// TIA Portal V20 export
// export: Created 2025-12-01T14:57:38.8034744Z, ExportSetting None, DisplayName Totally Integrated Automation Portal, DisplayVersion V20 Update 3, DisplayName TIA Portal Openness, DisplayVersion V20 Update 3, DisplayName TIA Portal Version Control Interface, DisplayVersion V20 Update 3, DisplayName STEP 7 Professional, DisplayVersion V20 Update 3, DisplayName STEP 7 Safety, DisplayVersion V20 Update 2, DisplayName WinCC Basic/Comfort/Advanced, DisplayVersion V20 Update 3, DisplayName WinCC Professional, DisplayVersion V20 Update 3, DisplayName WinCC Unified, DisplayVersion V20 Update 3
FUNCTION_BLOCK "FB75_MesaRodillos_PaletizadorCajasPlastico"   // FB75, LAD
TITLE = Mesa de Rodillos del DesPaletizador de Paletas
{ S7_Optimized_Access := 'FALSE' }
AUTHOR : PALETIZA
FAMILY : FRUTA
NAME : 20161001
VERSION : 1.0
// stored: AutoNumber false, SetENOAutomatically false
   VAR_INPUT
      Mesa : UInt;   // Mesa de la FB
      Error_Tx : Bool;   // Error en el Tx
      EnTension : Bool;   // Existe Tension en la Mesa
      Termico_Tx : Bool;   // Proteccion del Tx
      pHsMx : Bool;   // pHs de la Mesa
      pHsMx_PR1 : Bool;   // pHs de Protrusion de la Mesa. Nota: No existe >> ON
      Avance_Tx : Bool;   // Avance del Tx
      Retroceso_Tx : Bool;   // Retroceso del Tx
      Termico_MElev : Bool;   // Protecion de la Mesa Elevadora
      MElev_Abajo : Bool;   // Pos. Abajo >>> Mesa Elevadora
      MElev_Paleta : Bool;   // Pos. Paleta Normal >>> Mesa Elevadora
      MElev_EspacioBanda : Bool;   // Pos. Libre para mover la Banda >>> Mesa Elevadora
      ELEV_Bamper : Bool;   // Bamber >>> Mesa Elevadora
      MElev_EnMovimiento : Bool;   // En Movimiento >>> Mesa Elevadora
      PalaFija_IN : Bool;   // Pos. Cerrada >>> Pala Fija (Extendida)
      PalaFija_OUT : Bool;   // Pos. Abierta >>> Pala Fija (Recogida)
      PalaFija_EnMovimiento : Bool;   // En Movimiento >>> Pala Fija
      PalaMovil_IN : Bool;   // Pos. Cerrada >>> Pala Movil (Extendida)
      PalaMovil_OUT : Bool;   // Pos. Abierta >>> Pala Movil (Recogida)
      PalaMovil_EnMovimiento : Bool;   // En Movimiento >>> Pala Movil
      Centrador_IN : Bool;   // Pos. Sacado >>> Centrador
      Centrador_OUT : Bool;   // Pos. Recogido >>> Centrador
      Centrador_EnMovimiento : Bool;   // En Movimiento >>> Centrador
      Aviso_Paletizado : Bool;   // Aviso Paletizar >> Interlock Banda
      PermisoCierrePalas : Bool;   // Permiso Cierre de Palas >> Interlock Banda
      Permitir_AbrirPalas : Bool;   // Permiso DesPaletizar >> Interlock Banda
      Permitir_CerrarPalas : Bool;   // Permiso Abrir Palas >> Interlock Banda
      Permitir_AbrirCentrado : Bool;   // Permiso Abrir Centrador
      Permitir_CerrarCentrado : Bool;   // Permiso Cerrar Centrador
      MAnt_DescargaAct : Bool;   // E1 >> Mesa Anterior DescargaAct
      AVTF_MAnt_Mx : Bool;   // E1 >> Mesa Anterior AVTF
      P_Mens_MAnt_Mx : Bool;   // E1 >> Mesa Anterior P_Mens
      PTF_Mx_MSig : Bool;   // S1 >> Mesa Siguiente PTF
      FTF_Mx_MSig : Bool;   // S1 >> Mesa Siguiente FTF
      MSig_CargaAct : Bool;
      Mx_SimultaneoPaletizado : Bool;   // Config para Simultaneo de Paletizado
      Mx_VelocidadLenta_In : Bool;   // Forzar a Velociada Lenta
      F_EnvMens_Mx : Bool;   // Fin de Envio de Mensaje
      OrdSal_S01 : Bool;   // Orden de Salida por S1 (Paleta Cargada)
      V_CNT_pHsMx : Int := 500;   // Valor de Presencia
      V_CNTSeg_pHsMx : Int := 2000;   // Valor de Seguriadad para Presencia
      V_CNT_PasoLenta : Int := 2000;   // Valor de Paso a Lenta
      V_CNT_ApHsMx : Int := 500;   // Valor de Ausencia
      V_CNTSeg_ApHsMx : Int := 2000;   // Valor de Seguriadad para Ausencia
      V_TMP_EstablePalaMovil_IN : Int := 2000;   // TMP de Estabilidad de Pala Movil Extendida
      V_TOut_Tx_Mx : Int := 15000;   // TimeOut de Entrada por E1
      V_TOut_Palas : Int := 5000;   // TimeOut de las Palas
      V_TOut_Centrado : Int := 5000;   // TimeOut del Centrado
      V_TOut_MElevadora : Int := 10000;   // TimeOut de la Mesa Elevadora
      V_TMP_Protrusion : Int := 200;   // TMP de Protrusion
      V_CNT_PerdidapHs : Int := 1000;   // CNT de Perdida de pHs
   END_VAR
   VAR_OUTPUT
      P_EnvMens_PMx : Bool;   // Permiso de Enviar Mensaje de Presencia
      P_RecepOK_Mx : Bool;   // Recepcion OK
      Permiso_Paletizado : Bool;   // Permiso Paletizar >> Interlock Banda
      FinCierre_Palas : Bool;   // Fin Cierre Palas >> Interlock Banda
      PTF_MAnt_Mx : Bool;   // E1 >> Mesa Anterior PTF
      FTF_MAnt_Mx : Bool;   // E1 >> Mesa Anterior FTF
      AVTF_Mx_MSig : Bool;   // S1 >> Mesa Siguiente AVTF
      P_Mens_Mx_MSig : Bool;   // S1 >> Mesa Siguiente P_Mens
   END_VAR
   VAR
      Anular_prE1 : Bool;   // ???
      Anular_prS3 : Bool;   // ???
      Mx_ET00 : Bool;
      Mx_ET01 : Bool;
      Mx_ET02 : Bool;
      Mx_ET08 : Bool;
      Mx_ET09 : Bool;
      Mx_ET10 : Bool;
      Mx_ET11 : Bool;
      Mx_ET12 : Bool;
      Mx_ET13 : Bool;
      Mx_ET110 : Bool;
      Mx_ET111 : Bool;
      Mx_ET50 : Bool;
      Mx_ET51 : Bool;
      Mx_ET150 : Bool;
      Mx_ET151 : Bool;
      Mx_ET60 : Bool;
      Mx_ET61 : Bool;
      Mx_ET62 : Bool;
      Mx_ET63 : Bool;
      ProtocoloIniciado : Bool;   // Iniciado el Envio del Mensaje de Presencia
      PosMesa_OK : Bool;   // Posicion OK de la Mesa Elevadora
      SimultaneoPaletizado : Bool;   // Simultaneo Realizandose en el Paletizado
      Activar_OperativaPaletizado : Bool;   // Activar la Opertaiva de Simultaneo en el Paletizado
      CNT_pHsMx { S7_SetPoint := 'True'} : "FB910_CNT_UHS";   // CNT de la Presencia
      CNTSeg_pHsMx { S7_SetPoint := 'True'} : "FB910_CNT_UHS";   // CNT de Seguridad de la Presencia
      CNT_ApHsMx { S7_SetPoint := 'True'} : "FB910_CNT_UHS";   // CNT de la Ausencia
      CNTSeg_ApHsMx { S7_SetPoint := 'True'} : "FB910_CNT_UHS";   // CNT de Seguridad de la Ausencia
      TMP_EstablePalaMovil_IN { S7_SetPoint := 'True'} : "FB910_CNT_UHS";   // TMP de Estabilidad de Pala Movil Extendida
      TMP_EnTension { ExternalAccessible := 'False'; ExternalVisible := 'False'; ExternalWritable := 'False'; S7_SetPoint := 'True'} : "FB910_CNT_UHS";
      TOut_Av_Mx { S7_SetPoint := 'True'} : "FB910_CNT_UHS";   // Time Out de Entrada de E1
      TOut_MElevadora { S7_SetPoint := 'True'} : "FB910_CNT_UHS";   // Time Out de Recigida y Extension del Centrador
      TOut_Centrado { S7_SetPoint := 'True'} : "FB910_CNT_UHS";   // Time Out de Recigida y Extension de Pala Fija
      TOut_PalasFija { S7_SetPoint := 'True'} : "FB910_CNT_UHS";   // Time Out de Recigida y Extension de Pala Movil
      TOut_PalasMovil { S7_SetPoint := 'True'} : "FB910_CNT_UHS";   // Time Out de Subir y Bajar de la Mesa Elevadora
      TMP_Protrusion { S7_SetPoint := 'True'} : "FB910_CNT_UHS";   // TMP de la Protrusion
      CNT_PerdidapHs { S7_SetPoint := 'True'} : "FB910_CNT_UHS";   // CNT de Perdida de pHs
      STAT_EnvMens_PMx : Bool;   // Interna >> Envio del Mensaje de Presencia
      STAT_FTF_MAnt_Mx : Bool;   // Interna >> FTF de MAnt >> Mx
      STAT_AVTF_Mx_MSig : Bool;   // Interna >> AVTF de Mx >> MSig
      MA_Cerrar_Centrado : Bool;   // ????
      MA_Abrir_Centrado : Bool;   // ????
      MA_Abrir_PalasMovil : Bool;   // ????
      MA_Cerrar_PalasMovil : Bool;   // ????
      MA_Abrir_PalasFija : Bool;   // ????
      MA_Cerrar_PalasFija : Bool;   // ????
   END_VAR
   VAR_TEMP
      EstadoZona : "EstadoZona";   // Estado de Zona de la Mesa
      EstadoVI : "EstadosMesa";   // Estado del Vehiculo Inteliguente de la Mesa
      EstadoMAQ : "EstadoMaquina_MesaRodillos_PaletizadorCajasPlastico";   // Estado del Vehiculo Inteliguente de la Maquina
      ConfigFB : "UDT_ConfigFB";   // Configuracion de la FB de la Mesa
      V_Protrusion : Int;
      Aux_ET00 : Bool;
   END_VAR
BEGIN

REGION Network 1: Configuraciones Especiales
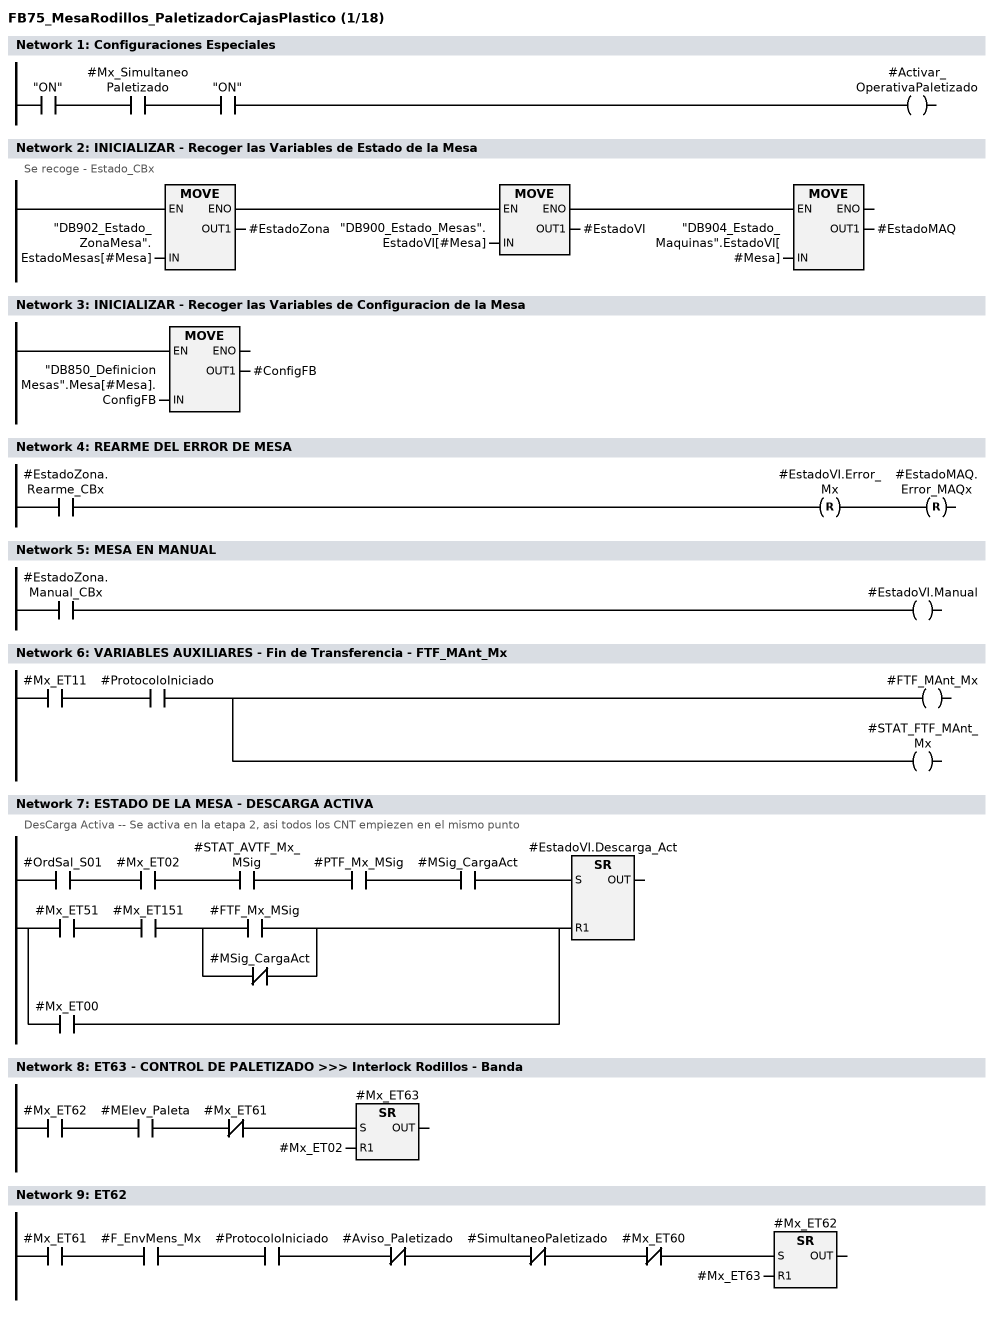
   RUNG wire#powerrail
      Contact( "ON" )
      Contact( #Mx_SimultaneoPaletizado )
      Contact( "ON" )
      Coil( #Activar_OperativaPaletizado )
   END_RUNG
   // the same network as SCL:
   #Activar_OperativaPaletizado := "ON" AND #Mx_SimultaneoPaletizado AND "ON";
END_REGION

REGION Network 2: INICIALIZAR - Recoger las Variables de Estado de la Mesa
   // Se recoge - Estado_CBx
   RUNG wire#powerrail
      Move(in := "DB902_Estado_ZonaMesa".EstadoMesas[#Mesa], out1 => #EstadoZona)
      Move(in := "DB900_Estado_Mesas".EstadoVI[#Mesa], out1 => #EstadoVI)
      Move(in := "DB904_Estado_Maquinas".EstadoVI[#Mesa], out1 => #EstadoMAQ)
   END_RUNG
   // the same network as SCL:
   #EstadoZona := "DB902_Estado_ZonaMesa".EstadoMesas[#Mesa];
   #EstadoVI := "DB900_Estado_Mesas".EstadoVI[#Mesa];
   #EstadoMAQ := "DB904_Estado_Maquinas".EstadoVI[#Mesa];
END_REGION

REGION Network 3: INICIALIZAR - Recoger las Variables de Configuracion de la Mesa
   RUNG wire#powerrail
      Move(in := "DB850_DefinicionMesas".Mesa[#Mesa].ConfigFB, out1 => #ConfigFB)
   END_RUNG
   // the same network as SCL:
   #ConfigFB := "DB850_DefinicionMesas".Mesa[#Mesa].ConfigFB;
END_REGION

REGION Network 4: REARME DEL ERROR DE MESA
   RUNG wire#powerrail
      Contact( #EstadoZona.Rearme_CBx )
      R_Coil( #EstadoVI.Error_Mx )
      R_Coil( #EstadoMAQ.Error_MAQx )
   END_RUNG
   // the same network as SCL:
   IF #EstadoZona.Rearme_CBx THEN
       #EstadoVI.Error_Mx := FALSE;
       #EstadoMAQ.Error_MAQx := FALSE;
   END_IF;
END_REGION

REGION Network 5: MESA EN MANUAL
   RUNG wire#powerrail
      Contact( #EstadoZona.Manual_CBx )
      Coil( #EstadoVI.Manual )
   END_RUNG
   // the same network as SCL:
   #EstadoVI.Manual := #EstadoZona.Manual_CBx;
END_REGION

REGION Network 6: VARIABLES AUXILIARES - Fin de Transferencia - FTF_MAnt_Mx
   RUNG wire#powerrail
      Contact( #Mx_ET11 )
      Contact( #ProtocoloIniciado )
      wire#w1
      Coil( #FTF_MAnt_Mx )
   END_RUNG
   RUNG wire#w1
      Coil( #STAT_FTF_MAnt_Mx )
   END_RUNG
   // the same network as SCL:
   #FTF_MAnt_Mx := #Mx_ET11 AND #ProtocoloIniciado;
   #STAT_FTF_MAnt_Mx := #FTF_MAnt_Mx;
END_REGION

REGION Network 7: ESTADO DE LA MESA - DESCARGA ACTIVA
   // DesCarga Activa -- Se activa en la etapa 2, asi todos los CNT empiezen en el mismo punto
   RUNG wire#powerrail
      Contact( #OrdSal_S01 )
      Contact( #Mx_ET02 )
      Contact( #STAT_AVTF_Mx_MSig )
      Contact( #PTF_Mx_MSig )
      Contact( #MSig_CargaAct )
      S_SR(operand := #EstadoVI.Descarga_Act, r1 := wire#w2)
   END_RUNG
   RUNG wire#powerrail
      Contact( #Mx_ET51 )
      Contact( #Mx_ET151 )
      wire#w1
      Contact( #FTF_Mx_MSig )
   END_RUNG wire#w2
   RUNG wire#w1
      I_Contact( #MSig_CargaAct )
   END_RUNG wire#w2
   RUNG wire#powerrail
      Contact( #Mx_ET00 )
   END_RUNG wire#w2
   // the same network as SCL:
   IF #OrdSal_S01 AND #Mx_ET02 AND #STAT_AVTF_Mx_MSig AND #PTF_Mx_MSig AND #MSig_CargaAct THEN
       #EstadoVI.Descarga_Act := TRUE;   // SR flip-flop
   END_IF;
   IF (#Mx_ET51 AND #Mx_ET151 AND (#FTF_Mx_MSig OR NOT #MSig_CargaAct)) OR #Mx_ET00 THEN
       #EstadoVI.Descarga_Act := FALSE;
   END_IF;
END_REGION

REGION Network 8: ET63 - CONTROL DE PALETIZADO >>> Interlock Rodillos - Banda
   RUNG wire#powerrail
      Contact( #Mx_ET62 )
      Contact( #MElev_Paleta )
      I_Contact( #Mx_ET61 )
      S_SR(operand := #Mx_ET63, r1 := #Mx_ET02)
   END_RUNG
   // the same network as SCL:
   IF #Mx_ET62 AND #MElev_Paleta AND NOT #Mx_ET61 THEN
       #Mx_ET63 := TRUE;   // SR flip-flop
   END_IF;
   IF #Mx_ET02 THEN #Mx_ET63 := FALSE; END_IF;
END_REGION

REGION Network 9: ET62
   RUNG wire#powerrail
      Contact( #Mx_ET61 )
      Contact( #F_EnvMens_Mx )
      Contact( #ProtocoloIniciado )
      I_Contact( #Aviso_Paletizado )
      I_Contact( #SimultaneoPaletizado )
      I_Contact( #Mx_ET60 )
      S_SR(operand := #Mx_ET62, r1 := #Mx_ET63)
   END_RUNG
   // the same network as SCL:
   IF #Mx_ET61 AND #F_EnvMens_Mx AND #ProtocoloIniciado AND NOT #Aviso_Paletizado AND NOT #SimultaneoPaletizado AND NOT #Mx_ET60 THEN
       #Mx_ET62 := TRUE;   // SR flip-flop
   END_IF;
   IF #Mx_ET63 THEN #Mx_ET62 := FALSE; END_IF;
END_REGION

REGION Network 10: ET61
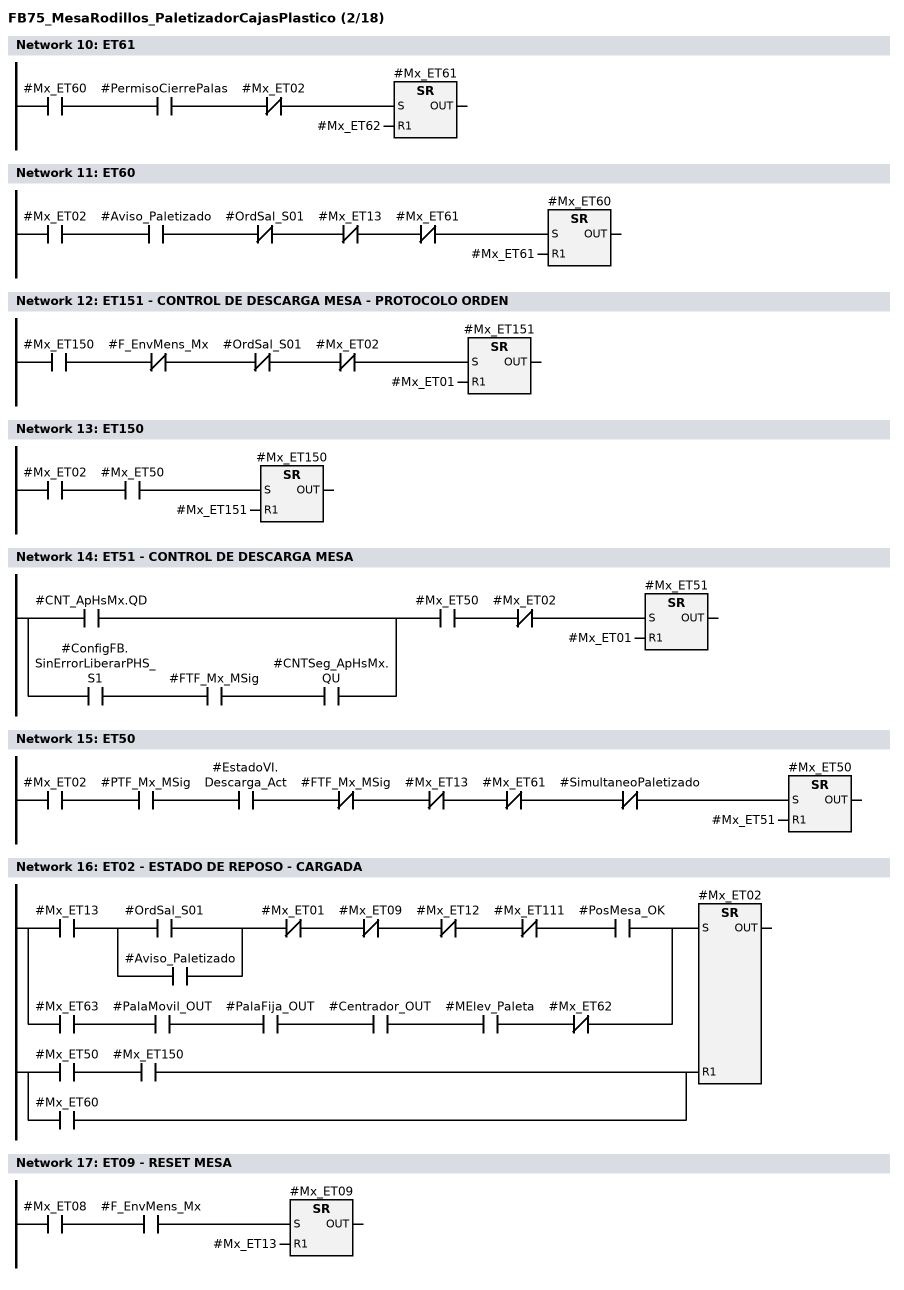
   RUNG wire#powerrail
      Contact( #Mx_ET60 )
      Contact( #PermisoCierrePalas )
      I_Contact( #Mx_ET02 )
      S_SR(operand := #Mx_ET61, r1 := #Mx_ET62)
   END_RUNG
   // the same network as SCL:
   IF #Mx_ET60 AND #PermisoCierrePalas AND NOT #Mx_ET02 THEN
       #Mx_ET61 := TRUE;   // SR flip-flop
   END_IF;
   IF #Mx_ET62 THEN #Mx_ET61 := FALSE; END_IF;
END_REGION

REGION Network 11: ET60
   RUNG wire#powerrail
      Contact( #Mx_ET02 )
      Contact( #Aviso_Paletizado )
      I_Contact( #OrdSal_S01 )
      I_Contact( #Mx_ET13 )
      I_Contact( #Mx_ET61 )
      S_SR(operand := #Mx_ET60, r1 := #Mx_ET61)
   END_RUNG
   // the same network as SCL:
   IF #Mx_ET02 AND #Aviso_Paletizado AND NOT #OrdSal_S01 AND NOT #Mx_ET13 AND NOT #Mx_ET61 THEN
       #Mx_ET60 := TRUE;   // SR flip-flop
   END_IF;
   IF #Mx_ET61 THEN #Mx_ET60 := FALSE; END_IF;
END_REGION

REGION Network 12: ET151 - CONTROL DE DESCARGA MESA - PROTOCOLO ORDEN
   RUNG wire#powerrail
      Contact( #Mx_ET150 )
      I_Contact( #F_EnvMens_Mx )
      I_Contact( #OrdSal_S01 )
      I_Contact( #Mx_ET02 )
      S_SR(operand := #Mx_ET151, r1 := #Mx_ET01)
   END_RUNG
   // the same network as SCL:
   IF #Mx_ET150 AND NOT #F_EnvMens_Mx AND NOT #OrdSal_S01 AND NOT #Mx_ET02 THEN
       #Mx_ET151 := TRUE;   // SR flip-flop
   END_IF;
   IF #Mx_ET01 THEN #Mx_ET151 := FALSE; END_IF;
END_REGION

REGION Network 13: ET150
   RUNG wire#powerrail
      Contact( #Mx_ET02 )
      Contact( #Mx_ET50 )
      S_SR(operand := #Mx_ET150, r1 := #Mx_ET151)
   END_RUNG
   // the same network as SCL:
   IF #Mx_ET02 AND #Mx_ET50 THEN
       #Mx_ET150 := TRUE;   // SR flip-flop
   END_IF;
   IF #Mx_ET151 THEN #Mx_ET150 := FALSE; END_IF;
END_REGION

REGION Network 14: ET51 - CONTROL DE DESCARGA MESA
   RUNG wire#powerrail
      Contact( #CNT_ApHsMx.QD )
      wire#w1
      Contact( #Mx_ET50 )
      I_Contact( #Mx_ET02 )
      S_SR(operand := #Mx_ET51, r1 := #Mx_ET01)
   END_RUNG
   RUNG wire#powerrail
      Contact( #ConfigFB.SinErrorLiberarPHS_S1 )
      Contact( #FTF_Mx_MSig )
      Contact( #CNTSeg_ApHsMx.QU )
   END_RUNG wire#w1
   // the same network as SCL:
   IF (#CNT_ApHsMx.QD OR (#ConfigFB.SinErrorLiberarPHS_S1 AND #FTF_Mx_MSig AND #CNTSeg_ApHsMx.QU)) AND #Mx_ET50 AND NOT #Mx_ET02 THEN
       #Mx_ET51 := TRUE;   // SR flip-flop
   END_IF;
   IF #Mx_ET01 THEN #Mx_ET51 := FALSE; END_IF;
END_REGION

REGION Network 15: ET50
   RUNG wire#powerrail
      Contact( #Mx_ET02 )
      Contact( #PTF_Mx_MSig )
      Contact( #EstadoVI.Descarga_Act )
      I_Contact( #FTF_Mx_MSig )
      I_Contact( #Mx_ET13 )
      I_Contact( #Mx_ET61 )
      I_Contact( #SimultaneoPaletizado )
      S_SR(operand := #Mx_ET50, r1 := #Mx_ET51)
   END_RUNG
   // the same network as SCL:
   IF #Mx_ET02 AND #PTF_Mx_MSig AND #EstadoVI.Descarga_Act AND NOT #FTF_Mx_MSig AND NOT #Mx_ET13 AND NOT #Mx_ET61 AND NOT #SimultaneoPaletizado THEN
       #Mx_ET50 := TRUE;   // SR flip-flop
   END_IF;
   IF #Mx_ET51 THEN #Mx_ET50 := FALSE; END_IF;
END_REGION

REGION Network 16: ET02 - ESTADO DE REPOSO - CARGADA
   RUNG wire#powerrail
      Contact( #Mx_ET13 )
      wire#w1
      Contact( #OrdSal_S01 )
      wire#w2
      I_Contact( #Mx_ET01 )
      I_Contact( #Mx_ET09 )
      I_Contact( #Mx_ET12 )
      I_Contact( #Mx_ET111 )
      Contact( #PosMesa_OK )
      wire#w3
      S_SR(operand := #Mx_ET02, r1 := wire#w4)
   END_RUNG
   RUNG wire#w1
      Contact( #Aviso_Paletizado )
   END_RUNG wire#w2
   RUNG wire#powerrail
      Contact( #Mx_ET63 )
      Contact( #PalaMovil_OUT )
      Contact( #PalaFija_OUT )
      Contact( #Centrador_OUT )
      Contact( #MElev_Paleta )
      I_Contact( #Mx_ET62 )
   END_RUNG wire#w3
   RUNG wire#powerrail
      Contact( #Mx_ET50 )
      Contact( #Mx_ET150 )
   END_RUNG wire#w4
   RUNG wire#powerrail
      Contact( #Mx_ET60 )
   END_RUNG wire#w4
   // the same network as SCL:
   IF (#Mx_ET13 AND (#OrdSal_S01 OR #Aviso_Paletizado) AND NOT #Mx_ET01 AND NOT #Mx_ET09 AND NOT #Mx_ET12 AND NOT #Mx_ET111 AND #PosMesa_OK) OR (#Mx_ET63 AND #PalaMovil_OUT AND #PalaFija_OUT AND #Centrador_OUT AND #MElev_Paleta AND NOT #Mx_ET62) THEN
       #Mx_ET02 := TRUE;   // SR flip-flop
   END_IF;
   IF (#Mx_ET50 AND #Mx_ET150) OR #Mx_ET60 THEN #Mx_ET02 := FALSE; END_IF;
END_REGION

REGION Network 17: ET09 - RESET MESA
   RUNG wire#powerrail
      Contact( #Mx_ET08 )
      Contact( #F_EnvMens_Mx )
      S_SR(operand := #Mx_ET09, r1 := #Mx_ET13)
   END_RUNG
   // the same network as SCL:
   IF #Mx_ET08 AND #F_EnvMens_Mx THEN
       #Mx_ET09 := TRUE;   // SR flip-flop
   END_IF;
   IF #Mx_ET13 THEN #Mx_ET09 := FALSE; END_IF;
END_REGION

REGION Network 18: ET08
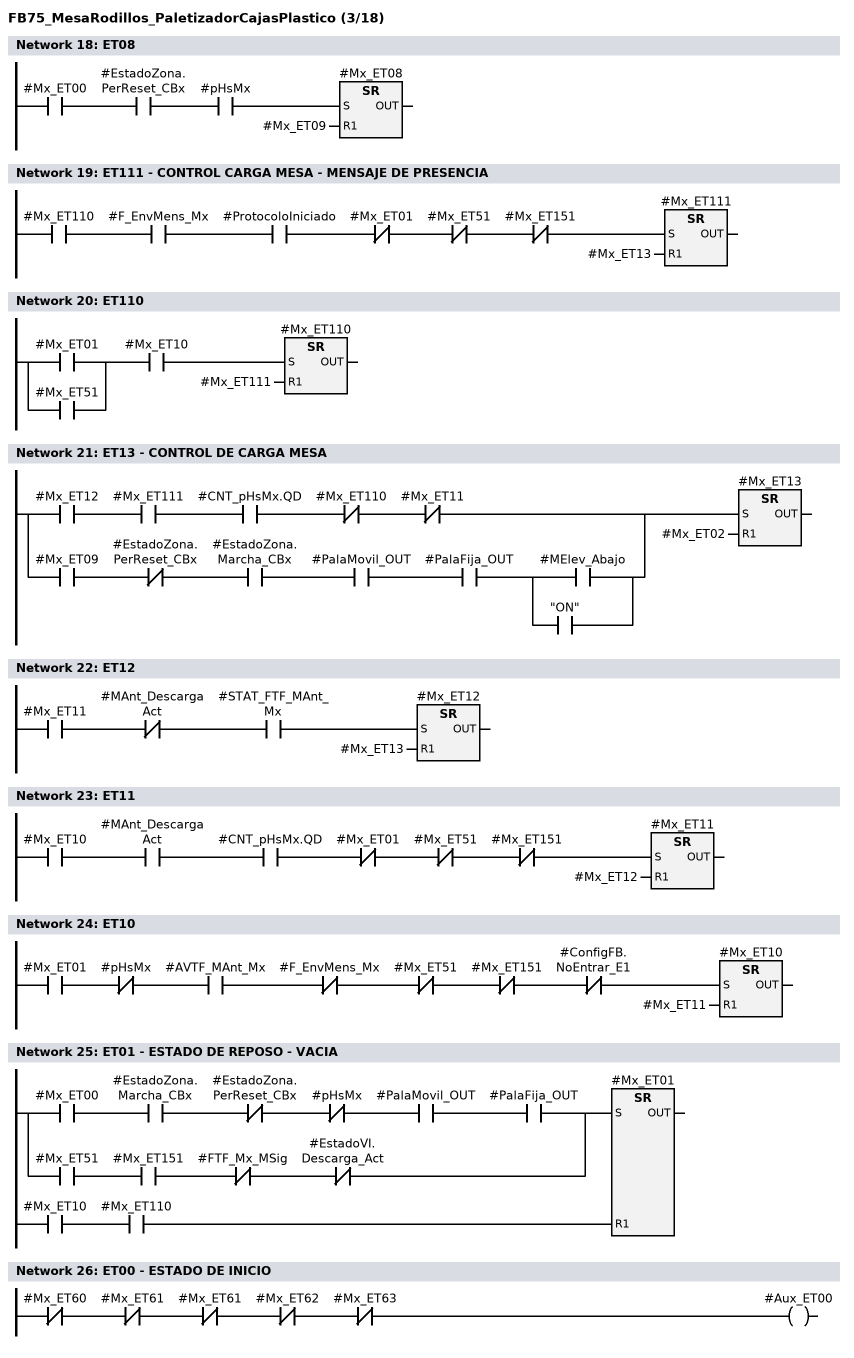
   RUNG wire#powerrail
      Contact( #Mx_ET00 )
      Contact( #EstadoZona.PerReset_CBx )
      Contact( #pHsMx )
      S_SR(operand := #Mx_ET08, r1 := #Mx_ET09)
   END_RUNG
   // the same network as SCL:
   IF #Mx_ET00 AND #EstadoZona.PerReset_CBx AND #pHsMx THEN
       #Mx_ET08 := TRUE;   // SR flip-flop
   END_IF;
   IF #Mx_ET09 THEN #Mx_ET08 := FALSE; END_IF;
END_REGION

REGION Network 19: ET111 - CONTROL CARGA MESA - MENSAJE DE PRESENCIA
   RUNG wire#powerrail
      Contact( #Mx_ET110 )
      Contact( #F_EnvMens_Mx )
      Contact( #ProtocoloIniciado )
      I_Contact( #Mx_ET01 )
      I_Contact( #Mx_ET51 )
      I_Contact( #Mx_ET151 )
      S_SR(operand := #Mx_ET111, r1 := #Mx_ET13)
   END_RUNG
   // the same network as SCL:
   IF #Mx_ET110 AND #F_EnvMens_Mx AND #ProtocoloIniciado AND NOT #Mx_ET01 AND NOT #Mx_ET51 AND NOT #Mx_ET151 THEN
       #Mx_ET111 := TRUE;   // SR flip-flop
   END_IF;
   IF #Mx_ET13 THEN #Mx_ET111 := FALSE; END_IF;
END_REGION

REGION Network 20: ET110
   RUNG wire#powerrail
      Contact( #Mx_ET01 )
      wire#w1
      Contact( #Mx_ET10 )
      S_SR(operand := #Mx_ET110, r1 := #Mx_ET111)
   END_RUNG
   RUNG wire#powerrail
      Contact( #Mx_ET51 )
   END_RUNG wire#w1
   // the same network as SCL:
   IF (#Mx_ET01 OR #Mx_ET51) AND #Mx_ET10 THEN
       #Mx_ET110 := TRUE;   // SR flip-flop
   END_IF;
   IF #Mx_ET111 THEN #Mx_ET110 := FALSE; END_IF;
END_REGION

REGION Network 21: ET13 - CONTROL DE CARGA MESA
   RUNG wire#powerrail
      Contact( #Mx_ET12 )
      Contact( #Mx_ET111 )
      Contact( #CNT_pHsMx.QD )
      I_Contact( #Mx_ET110 )
      I_Contact( #Mx_ET11 )
      wire#w1
      S_SR(operand := #Mx_ET13, r1 := #Mx_ET02)
   END_RUNG
   RUNG wire#powerrail
      Contact( #Mx_ET09 )
      I_Contact( #EstadoZona.PerReset_CBx )
      Contact( #EstadoZona.Marcha_CBx )
      Contact( #PalaMovil_OUT )
      Contact( #PalaFija_OUT )
      wire#w2
      Contact( #MElev_Abajo )
   END_RUNG wire#w1
   RUNG wire#w2
      Contact( "ON" )
   END_RUNG wire#w1
   // the same network as SCL:
   IF (#Mx_ET12 AND #Mx_ET111 AND #CNT_pHsMx.QD AND NOT #Mx_ET110 AND NOT #Mx_ET11) OR (#Mx_ET09 AND NOT #EstadoZona.PerReset_CBx AND #EstadoZona.Marcha_CBx AND #PalaMovil_OUT AND #PalaFija_OUT AND (#MElev_Abajo OR "ON")) THEN
       #Mx_ET13 := TRUE;   // SR flip-flop
   END_IF;
   IF #Mx_ET02 THEN #Mx_ET13 := FALSE; END_IF;
END_REGION

REGION Network 22: ET12
   RUNG wire#powerrail
      Contact( #Mx_ET11 )
      I_Contact( #MAnt_DescargaAct )
      Contact( #STAT_FTF_MAnt_Mx )
      S_SR(operand := #Mx_ET12, r1 := #Mx_ET13)
   END_RUNG
   // the same network as SCL:
   IF #Mx_ET11 AND NOT #MAnt_DescargaAct AND #STAT_FTF_MAnt_Mx THEN
       #Mx_ET12 := TRUE;   // SR flip-flop
   END_IF;
   IF #Mx_ET13 THEN #Mx_ET12 := FALSE; END_IF;
END_REGION

REGION Network 23: ET11
   RUNG wire#powerrail
      Contact( #Mx_ET10 )
      Contact( #MAnt_DescargaAct )
      Contact( #CNT_pHsMx.QD )
      I_Contact( #Mx_ET01 )
      I_Contact( #Mx_ET51 )
      I_Contact( #Mx_ET151 )
      S_SR(operand := #Mx_ET11, r1 := #Mx_ET12)
   END_RUNG
   // the same network as SCL:
   IF #Mx_ET10 AND #MAnt_DescargaAct AND #CNT_pHsMx.QD AND NOT #Mx_ET01 AND NOT #Mx_ET51 AND NOT #Mx_ET151 THEN
       #Mx_ET11 := TRUE;   // SR flip-flop
   END_IF;
   IF #Mx_ET12 THEN #Mx_ET11 := FALSE; END_IF;
END_REGION

REGION Network 24: ET10
   RUNG wire#powerrail
      Contact( #Mx_ET01 )
      I_Contact( #pHsMx )
      Contact( #AVTF_MAnt_Mx )
      I_Contact( #F_EnvMens_Mx )
      I_Contact( #Mx_ET51 )
      I_Contact( #Mx_ET151 )
      I_Contact( #ConfigFB.NoEntrar_E1 )
      S_SR(operand := #Mx_ET10, r1 := #Mx_ET11)
   END_RUNG
   // the same network as SCL:
   IF #Mx_ET01 AND NOT #pHsMx AND #AVTF_MAnt_Mx AND NOT #F_EnvMens_Mx AND NOT #Mx_ET51 AND NOT #Mx_ET151 AND NOT #ConfigFB.NoEntrar_E1 THEN
       #Mx_ET10 := TRUE;   // SR flip-flop
   END_IF;
   IF #Mx_ET11 THEN #Mx_ET10 := FALSE; END_IF;
END_REGION

REGION Network 25: ET01 - ESTADO DE REPOSO - VACIA
   RUNG wire#powerrail
      Contact( #Mx_ET00 )
      Contact( #EstadoZona.Marcha_CBx )
      I_Contact( #EstadoZona.PerReset_CBx )
      I_Contact( #pHsMx )
      Contact( #PalaMovil_OUT )
      Contact( #PalaFija_OUT )
      wire#w1
      S_SR(operand := #Mx_ET01, r1 := wire#w2)
   END_RUNG
   RUNG wire#powerrail
      Contact( #Mx_ET51 )
      Contact( #Mx_ET151 )
      I_Contact( #FTF_Mx_MSig )
      I_Contact( #EstadoVI.Descarga_Act )
   END_RUNG wire#w1
   RUNG wire#powerrail
      Contact( #Mx_ET10 )
      Contact( #Mx_ET110 )
   END_RUNG wire#w2
   // the same network as SCL:
   IF (#Mx_ET00 AND #EstadoZona.Marcha_CBx AND NOT #EstadoZona.PerReset_CBx AND NOT #pHsMx AND #PalaMovil_OUT AND #PalaFija_OUT) OR (#Mx_ET51 AND #Mx_ET151 AND NOT #FTF_Mx_MSig AND NOT #EstadoVI.Descarga_Act) THEN
       #Mx_ET01 := TRUE;   // SR flip-flop
   END_IF;
   IF #Mx_ET10 AND #Mx_ET110 THEN #Mx_ET01 := FALSE; END_IF;
END_REGION

REGION Network 26: ET00 - ESTADO DE INICIO
   RUNG wire#powerrail
      I_Contact( #Mx_ET60 )
      I_Contact( #Mx_ET61 )
      I_Contact( #Mx_ET61 )
      I_Contact( #Mx_ET62 )
      I_Contact( #Mx_ET63 )
      Coil( #Aux_ET00 )
   END_RUNG
   // the same network as SCL:
   #Aux_ET00 := NOT #Mx_ET60 AND NOT #Mx_ET61 AND NOT #Mx_ET61 AND NOT #Mx_ET62 AND NOT #Mx_ET63;
END_REGION

REGION Network 27: ---
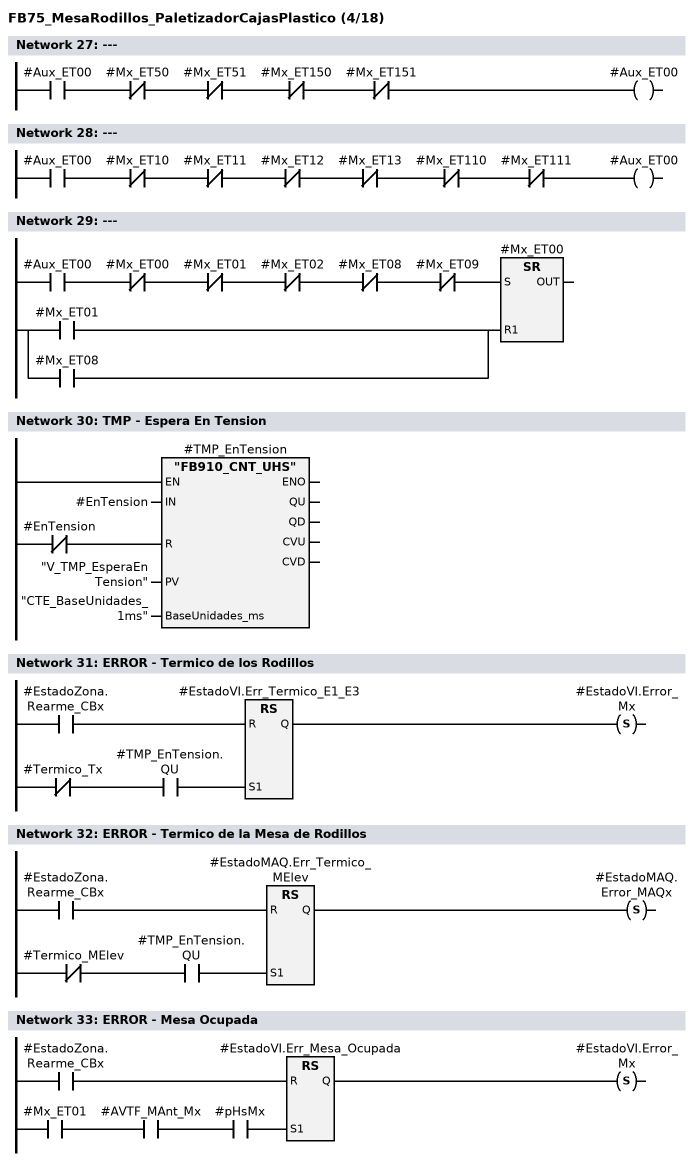
   RUNG wire#powerrail
      Contact( #Aux_ET00 )
      I_Contact( #Mx_ET50 )
      I_Contact( #Mx_ET51 )
      I_Contact( #Mx_ET150 )
      I_Contact( #Mx_ET151 )
      Coil( #Aux_ET00 )
   END_RUNG
   // the same network as SCL:
   #Aux_ET00 := #Aux_ET00 AND NOT #Mx_ET50 AND NOT #Mx_ET51 AND NOT #Mx_ET150 AND NOT #Mx_ET151;
END_REGION

REGION Network 28: ---
   RUNG wire#powerrail
      Contact( #Aux_ET00 )
      I_Contact( #Mx_ET10 )
      I_Contact( #Mx_ET11 )
      I_Contact( #Mx_ET12 )
      I_Contact( #Mx_ET13 )
      I_Contact( #Mx_ET110 )
      I_Contact( #Mx_ET111 )
      Coil( #Aux_ET00 )
   END_RUNG
   // the same network as SCL:
   #Aux_ET00 := #Aux_ET00 AND NOT #Mx_ET10 AND NOT #Mx_ET11 AND NOT #Mx_ET12 AND NOT #Mx_ET13 AND NOT #Mx_ET110 AND NOT #Mx_ET111;
END_REGION

REGION Network 29: ---
   RUNG wire#powerrail
      Contact( #Aux_ET00 )
      I_Contact( #Mx_ET00 )
      I_Contact( #Mx_ET01 )
      I_Contact( #Mx_ET02 )
      I_Contact( #Mx_ET08 )
      I_Contact( #Mx_ET09 )
      S_SR(operand := #Mx_ET00, r1 := wire#w1)
   END_RUNG
   RUNG wire#powerrail
      Contact( #Mx_ET01 )
   END_RUNG wire#w1
   RUNG wire#powerrail
      Contact( #Mx_ET08 )
   END_RUNG wire#w1
   // the same network as SCL:
   IF #Aux_ET00 AND NOT #Mx_ET00 AND NOT #Mx_ET01 AND NOT #Mx_ET02 AND NOT #Mx_ET08 AND NOT #Mx_ET09 THEN
       #Mx_ET00 := TRUE;   // SR flip-flop
   END_IF;
   IF #Mx_ET01 OR #Mx_ET08 THEN #Mx_ET00 := FALSE; END_IF;
END_REGION

REGION Network 30: TMP - Espera En Tension
   RUNG wire#powerrail
      #TMP_EnTension(R := wire#w1, IN := #EnTension, PV := "V_TMP_EsperaEnTension", BaseUnidades_ms := "CTE_BaseUnidades_1ms", QU =>, QD =>, CVU =>, CVD =>)
   END_RUNG
   RUNG wire#powerrail
      I_Contact( #EnTension )
   END_RUNG wire#w1
   // the same network as SCL:
   #TMP_EnTension(IN := #EnTension,   // "FB910_CNT_UHS"
                  R := NOT #EnTension,
                  PV := "V_TMP_EsperaEnTension",
                  BaseUnidades_ms := "CTE_BaseUnidades_1ms");
END_REGION

REGION Network 31: ERROR - Termico de los Rodillos
   RUNG wire#powerrail
      Contact( #EstadoZona.Rearme_CBx )
      S_RS(operand := #EstadoVI.Err_Termico_E1_E3, s1 := wire#w1)
      S_Coil( #EstadoVI.Error_Mx )
   END_RUNG
   RUNG wire#powerrail
      I_Contact( #Termico_Tx )
      Contact( #TMP_EnTension.QU )
   END_RUNG wire#w1
   // the same network as SCL:
   IF #EstadoZona.Rearme_CBx THEN
       #EstadoVI.Err_Termico_E1_E3 := FALSE;   // RS flip-flop
   END_IF;
   IF NOT #Termico_Tx AND #TMP_EnTension.QU THEN #EstadoVI.Err_Termico_E1_E3 := TRUE; END_IF;
   IF #EstadoVI.Err_Termico_E1_E3 THEN #EstadoVI.Error_Mx := TRUE; END_IF;
END_REGION

REGION Network 32: ERROR - Termico de la Mesa de Rodillos
   RUNG wire#powerrail
      Contact( #EstadoZona.Rearme_CBx )
      S_RS(operand := #EstadoMAQ.Err_Termico_MElev, s1 := wire#w1)
      S_Coil( #EstadoMAQ.Error_MAQx )
   END_RUNG
   RUNG wire#powerrail
      I_Contact( #Termico_MElev )
      Contact( #TMP_EnTension.QU )
   END_RUNG wire#w1
   // the same network as SCL:
   IF #EstadoZona.Rearme_CBx THEN
       #EstadoMAQ.Err_Termico_MElev := FALSE;   // RS flip-flop
   END_IF;
   IF NOT #Termico_MElev AND #TMP_EnTension.QU THEN #EstadoMAQ.Err_Termico_MElev := TRUE; END_IF;
   IF #EstadoMAQ.Err_Termico_MElev THEN #EstadoMAQ.Error_MAQx := TRUE; END_IF;
END_REGION

REGION Network 33: ERROR - Mesa Ocupada
   RUNG wire#powerrail
      Contact( #EstadoZona.Rearme_CBx )
      S_RS(operand := #EstadoVI.Err_Mesa_Ocupada, s1 := wire#w1)
      S_Coil( #EstadoVI.Error_Mx )
   END_RUNG
   RUNG wire#powerrail
      Contact( #Mx_ET01 )
      Contact( #AVTF_MAnt_Mx )
      Contact( #pHsMx )
   END_RUNG wire#w1
   // the same network as SCL:
   IF #EstadoZona.Rearme_CBx THEN
       #EstadoVI.Err_Mesa_Ocupada := FALSE;   // RS flip-flop
   END_IF;
   IF #Mx_ET01 AND #AVTF_MAnt_Mx AND #pHsMx THEN #EstadoVI.Err_Mesa_Ocupada := TRUE; END_IF;
   IF #EstadoVI.Err_Mesa_Ocupada THEN #EstadoVI.Error_Mx := TRUE; END_IF;
END_REGION

REGION Network 34: CNT - ERROR - Arrastre
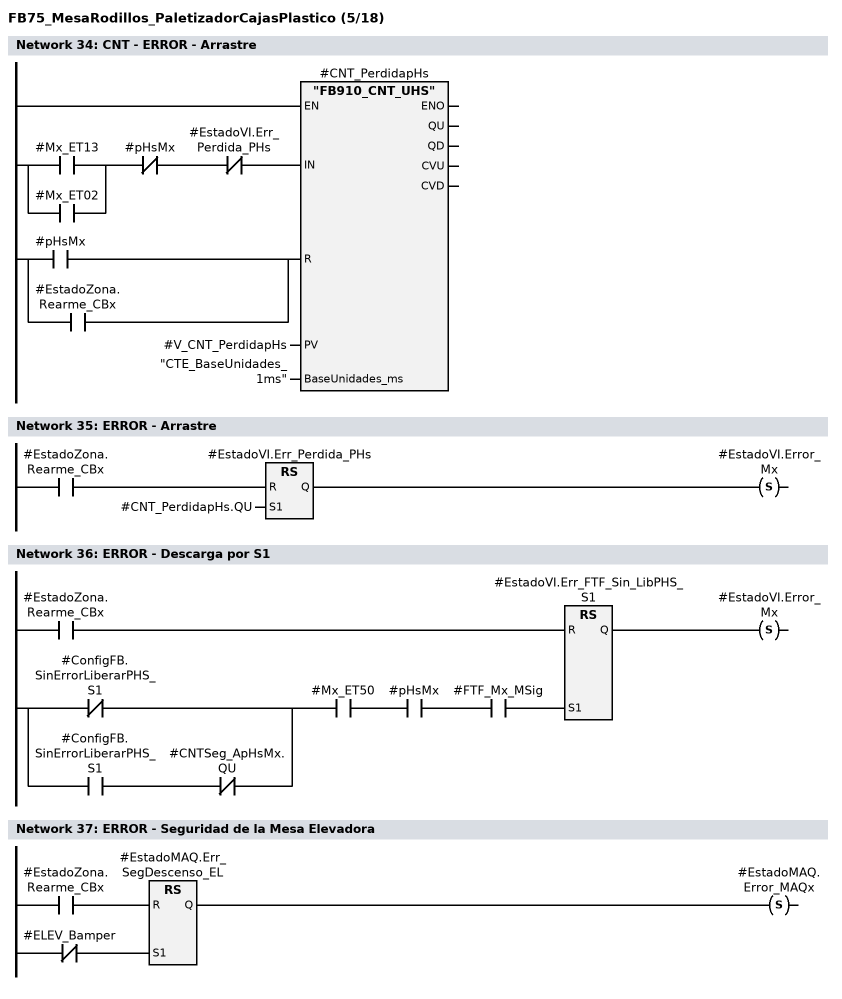
   RUNG wire#powerrail
      #CNT_PerdidapHs(IN := wire#w2, R := wire#w3, PV := #V_CNT_PerdidapHs, BaseUnidades_ms := "CTE_BaseUnidades_1ms", QU =>, QD =>, CVU =>, CVD =>)
   END_RUNG
   RUNG wire#powerrail
      Contact( #Mx_ET13 )
      wire#w1
      I_Contact( #pHsMx )
      I_Contact( #EstadoVI.Err_Perdida_PHs )
   END_RUNG wire#w2
   RUNG wire#powerrail
      Contact( #Mx_ET02 )
   END_RUNG wire#w1
   RUNG wire#powerrail
      Contact( #pHsMx )
   END_RUNG wire#w3
   RUNG wire#powerrail
      Contact( #EstadoZona.Rearme_CBx )
   END_RUNG wire#w3
   // the same network as SCL:
   #CNT_PerdidapHs(IN := (#Mx_ET13 OR #Mx_ET02) AND NOT #pHsMx AND NOT #EstadoVI.Err_Perdida_PHs,   // "FB910_CNT_UHS"
                   R := #pHsMx OR #EstadoZona.Rearme_CBx,
                   PV := #V_CNT_PerdidapHs,
                   BaseUnidades_ms := "CTE_BaseUnidades_1ms");
END_REGION

REGION Network 35: ERROR - Arrastre
   RUNG wire#powerrail
      Contact( #EstadoZona.Rearme_CBx )
      S_RS(operand := #EstadoVI.Err_Perdida_PHs, s1 := #CNT_PerdidapHs.QU)
      S_Coil( #EstadoVI.Error_Mx )
   END_RUNG
   // the same network as SCL:
   IF #EstadoZona.Rearme_CBx THEN
       #EstadoVI.Err_Perdida_PHs := FALSE;   // RS flip-flop
   END_IF;
   IF #CNT_PerdidapHs.QU THEN #EstadoVI.Err_Perdida_PHs := TRUE; END_IF;
   IF #EstadoVI.Err_Perdida_PHs THEN #EstadoVI.Error_Mx := TRUE; END_IF;
END_REGION

REGION Network 36: ERROR - Descarga por S1
   RUNG wire#powerrail
      Contact( #EstadoZona.Rearme_CBx )
      S_RS(operand := #EstadoVI.Err_FTF_Sin_LibPHS_S1, s1 := wire#w2)
      S_Coil( #EstadoVI.Error_Mx )
   END_RUNG
   RUNG wire#powerrail
      I_Contact( #ConfigFB.SinErrorLiberarPHS_S1 )
      wire#w1
      Contact( #Mx_ET50 )
      Contact( #pHsMx )
      Contact( #FTF_Mx_MSig )
   END_RUNG wire#w2
   RUNG wire#powerrail
      Contact( #ConfigFB.SinErrorLiberarPHS_S1 )
      I_Contact( #CNTSeg_ApHsMx.QU )
   END_RUNG wire#w1
   // the same network as SCL:
   IF #EstadoZona.Rearme_CBx THEN
       #EstadoVI.Err_FTF_Sin_LibPHS_S1 := FALSE;   // RS flip-flop
   END_IF;
   IF (NOT #ConfigFB.SinErrorLiberarPHS_S1 OR (#ConfigFB.SinErrorLiberarPHS_S1 AND NOT #CNTSeg_ApHsMx.QU)) AND #Mx_ET50 AND #pHsMx AND #FTF_Mx_MSig THEN
       #EstadoVI.Err_FTF_Sin_LibPHS_S1 := TRUE;
   END_IF;
   IF #EstadoVI.Err_FTF_Sin_LibPHS_S1 THEN #EstadoVI.Error_Mx := TRUE; END_IF;
END_REGION

REGION Network 37: ERROR - Seguridad de la Mesa Elevadora
   RUNG wire#powerrail
      Contact( #EstadoZona.Rearme_CBx )
      S_RS(operand := #EstadoMAQ.Err_SegDescenso_EL, s1 := wire#w1)
      S_Coil( #EstadoMAQ.Error_MAQx )
   END_RUNG
   RUNG wire#powerrail
      I_Contact( #ELEV_Bamper )
   END_RUNG wire#w1
   // the same network as SCL:
   IF #EstadoZona.Rearme_CBx THEN
       #EstadoMAQ.Err_SegDescenso_EL := FALSE;   // RS flip-flop
   END_IF;
   IF NOT #ELEV_Bamper THEN #EstadoMAQ.Err_SegDescenso_EL := TRUE; END_IF;
   IF #EstadoMAQ.Err_SegDescenso_EL THEN #EstadoMAQ.Error_MAQx := TRUE; END_IF;
END_REGION

REGION Network 38: TMP - ERROR - TimeOut Avance
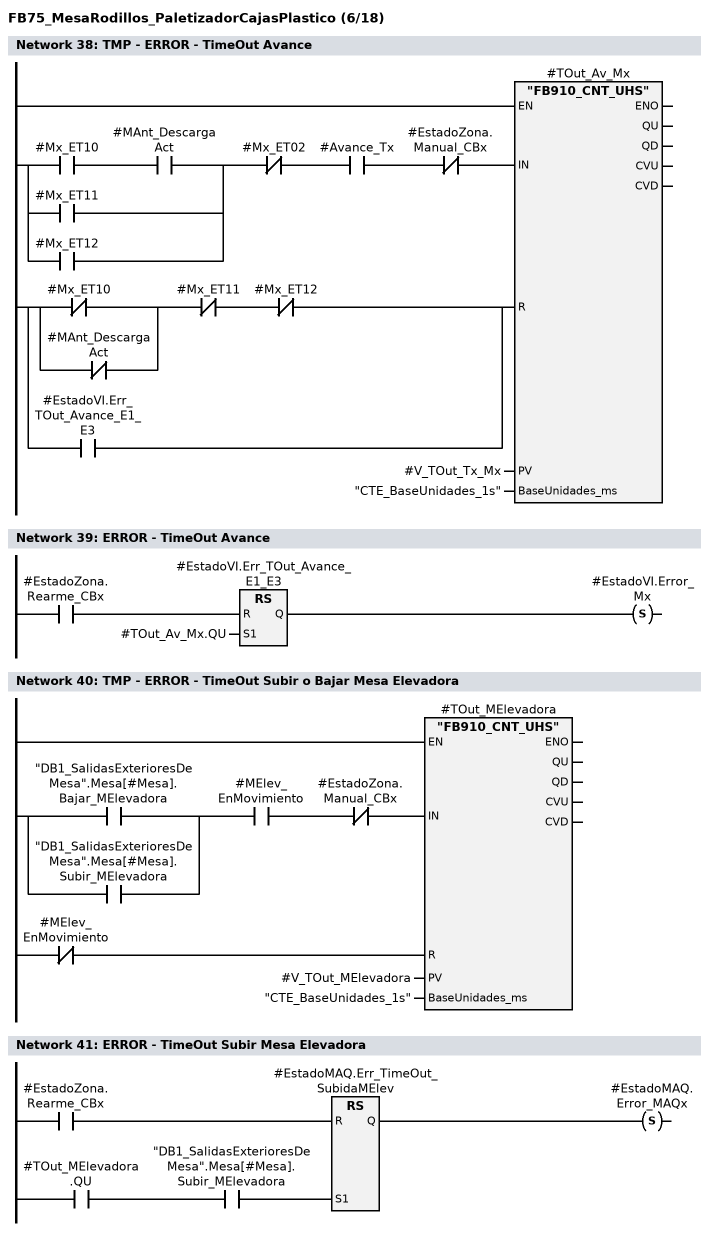
   RUNG wire#powerrail
      #TOut_Av_Mx(IN := wire#w2, R := wire#w4, PV := #V_TOut_Tx_Mx, BaseUnidades_ms := "CTE_BaseUnidades_1s", QU =>, QD =>, CVU =>, CVD =>)
   END_RUNG
   RUNG wire#powerrail
      Contact( #Mx_ET10 )
      Contact( #MAnt_DescargaAct )
      wire#w1
      I_Contact( #Mx_ET02 )
      Contact( #Avance_Tx )
      I_Contact( #EstadoZona.Manual_CBx )
   END_RUNG wire#w2
   RUNG wire#powerrail
      Contact( #Mx_ET11 )
   END_RUNG wire#w1
   RUNG wire#powerrail
      Contact( #Mx_ET12 )
   END_RUNG wire#w1
   RUNG wire#powerrail
      I_Contact( #Mx_ET10 )
      wire#w3
      I_Contact( #Mx_ET11 )
      I_Contact( #Mx_ET12 )
   END_RUNG wire#w4
   RUNG wire#powerrail
      I_Contact( #MAnt_DescargaAct )
   END_RUNG wire#w3
   RUNG wire#powerrail
      Contact( #EstadoVI.Err_TOut_Avance_E1_E3 )
   END_RUNG wire#w4
   // the same network as SCL:
   #TOut_Av_Mx(IN := ((#Mx_ET10 AND #MAnt_DescargaAct) OR #Mx_ET11 OR #Mx_ET12) AND NOT #Mx_ET02 AND #Avance_Tx AND NOT #EstadoZona.Manual_CBx,   // "FB910_CNT_UHS"
               R := ((NOT #Mx_ET10 OR NOT #MAnt_DescargaAct) AND NOT #Mx_ET11 AND NOT #Mx_ET12) OR #EstadoVI.Err_TOut_Avance_E1_E3,
               PV := #V_TOut_Tx_Mx,
               BaseUnidades_ms := "CTE_BaseUnidades_1s");
END_REGION

REGION Network 39: ERROR - TimeOut Avance
   RUNG wire#powerrail
      Contact( #EstadoZona.Rearme_CBx )
      S_RS(operand := #EstadoVI.Err_TOut_Avance_E1_E3, s1 := #TOut_Av_Mx.QU)
      S_Coil( #EstadoVI.Error_Mx )
   END_RUNG
   // the same network as SCL:
   IF #EstadoZona.Rearme_CBx THEN
       #EstadoVI.Err_TOut_Avance_E1_E3 := FALSE;   // RS flip-flop
   END_IF;
   IF #TOut_Av_Mx.QU THEN #EstadoVI.Err_TOut_Avance_E1_E3 := TRUE; END_IF;
   IF #EstadoVI.Err_TOut_Avance_E1_E3 THEN #EstadoVI.Error_Mx := TRUE; END_IF;
END_REGION

REGION Network 40: TMP - ERROR - TimeOut Subir o Bajar Mesa Elevadora
   RUNG wire#powerrail
      #TOut_MElevadora(IN := wire#w2, R := wire#w3, PV := #V_TOut_MElevadora, BaseUnidades_ms := "CTE_BaseUnidades_1s", QU =>, QD =>, CVU =>, CVD =>)
   END_RUNG
   RUNG wire#powerrail
      Contact( "DB1_SalidasExterioresDeMesa".Mesa[#Mesa].Bajar_MElevadora )
      wire#w1
      Contact( #MElev_EnMovimiento )
      I_Contact( #EstadoZona.Manual_CBx )
   END_RUNG wire#w2
   RUNG wire#powerrail
      Contact( "DB1_SalidasExterioresDeMesa".Mesa[#Mesa].Subir_MElevadora )
   END_RUNG wire#w1
   RUNG wire#powerrail
      I_Contact( #MElev_EnMovimiento )
   END_RUNG wire#w3
   // the same network as SCL:
   #TOut_MElevadora(IN := ("DB1_SalidasExterioresDeMesa".Mesa[#Mesa].Bajar_MElevadora OR "DB1_SalidasExterioresDeMesa".Mesa[#Mesa].Subir_MElevadora) AND #MElev_EnMovimiento AND NOT #EstadoZona.Manual_CBx,   // "FB910_CNT_UHS"
                    R := NOT #MElev_EnMovimiento,
                    PV := #V_TOut_MElevadora,
                    BaseUnidades_ms := "CTE_BaseUnidades_1s");
END_REGION

REGION Network 41: ERROR - TimeOut Subir Mesa Elevadora
   RUNG wire#powerrail
      Contact( #EstadoZona.Rearme_CBx )
      S_RS(operand := #EstadoMAQ.Err_TimeOut_SubidaMElev, s1 := wire#w1)
      S_Coil( #EstadoMAQ.Error_MAQx )
   END_RUNG
   RUNG wire#powerrail
      Contact( #TOut_MElevadora.QU )
      Contact( "DB1_SalidasExterioresDeMesa".Mesa[#Mesa].Subir_MElevadora )
   END_RUNG wire#w1
   // the same network as SCL:
   IF #EstadoZona.Rearme_CBx THEN
       #EstadoMAQ.Err_TimeOut_SubidaMElev := FALSE;   // RS flip-flop
   END_IF;
   IF #TOut_MElevadora.QU AND "DB1_SalidasExterioresDeMesa".Mesa[#Mesa].Subir_MElevadora THEN
       #EstadoMAQ.Err_TimeOut_SubidaMElev := TRUE;
   END_IF;
   IF #EstadoMAQ.Err_TimeOut_SubidaMElev THEN #EstadoMAQ.Error_MAQx := TRUE; END_IF;
END_REGION

REGION Network 42: ERROR - TimeOut Bajar Mesa Elevadora
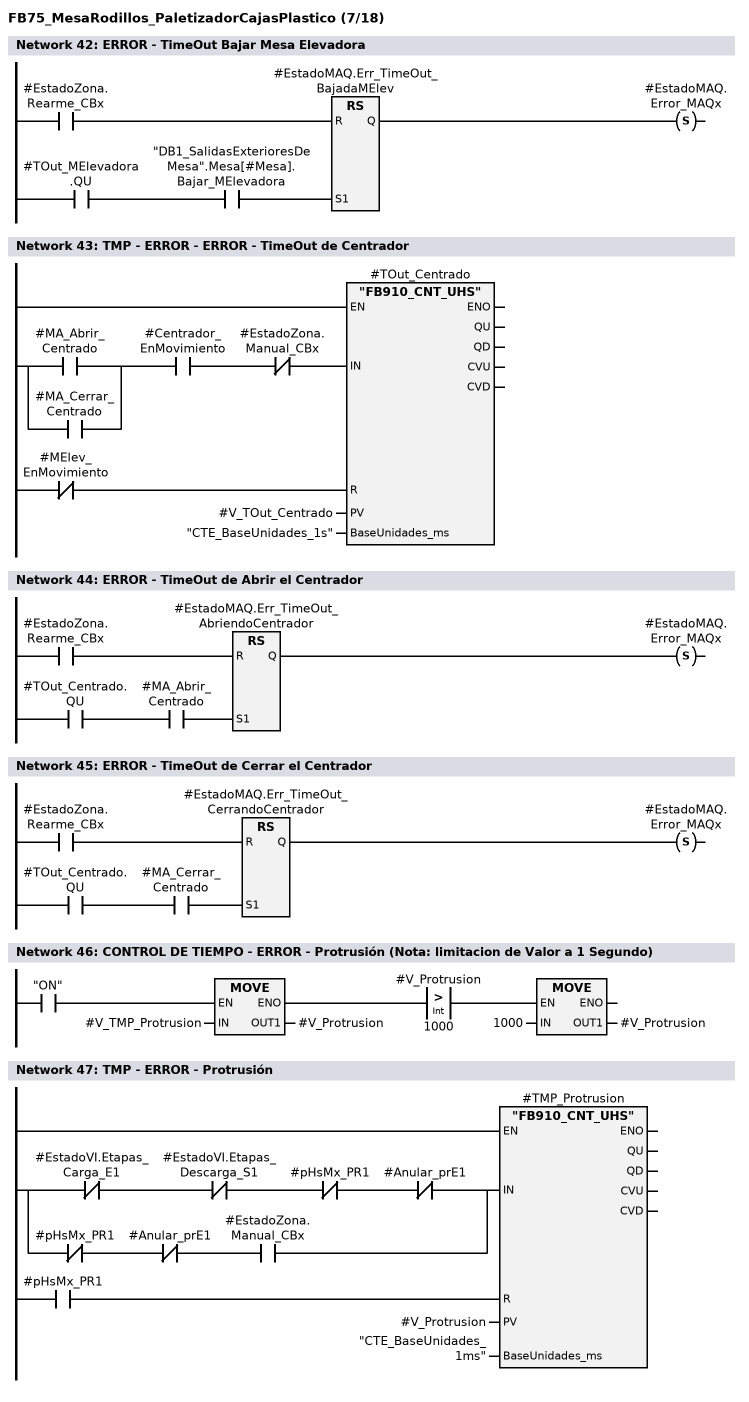
   RUNG wire#powerrail
      Contact( #EstadoZona.Rearme_CBx )
      S_RS(operand := #EstadoMAQ.Err_TimeOut_BajadaMElev, s1 := wire#w1)
      S_Coil( #EstadoMAQ.Error_MAQx )
   END_RUNG
   RUNG wire#powerrail
      Contact( #TOut_MElevadora.QU )
      Contact( "DB1_SalidasExterioresDeMesa".Mesa[#Mesa].Bajar_MElevadora )
   END_RUNG wire#w1
   // the same network as SCL:
   IF #EstadoZona.Rearme_CBx THEN
       #EstadoMAQ.Err_TimeOut_BajadaMElev := FALSE;   // RS flip-flop
   END_IF;
   IF #TOut_MElevadora.QU AND "DB1_SalidasExterioresDeMesa".Mesa[#Mesa].Bajar_MElevadora THEN
       #EstadoMAQ.Err_TimeOut_BajadaMElev := TRUE;
   END_IF;
   IF #EstadoMAQ.Err_TimeOut_BajadaMElev THEN #EstadoMAQ.Error_MAQx := TRUE; END_IF;
END_REGION

REGION Network 43: TMP - ERROR - ERROR - TimeOut de Centrador
   RUNG wire#powerrail
      #TOut_Centrado(IN := wire#w2, R := wire#w3, PV := #V_TOut_Centrado, BaseUnidades_ms := "CTE_BaseUnidades_1s", QU =>, QD =>, CVU =>, CVD =>)
   END_RUNG
   RUNG wire#powerrail
      Contact( #MA_Abrir_Centrado )
      wire#w1
      Contact( #Centrador_EnMovimiento )
      I_Contact( #EstadoZona.Manual_CBx )
   END_RUNG wire#w2
   RUNG wire#powerrail
      Contact( #MA_Cerrar_Centrado )
   END_RUNG wire#w1
   RUNG wire#powerrail
      I_Contact( #MElev_EnMovimiento )
   END_RUNG wire#w3
   // the same network as SCL:
   #TOut_Centrado(IN := (#MA_Abrir_Centrado OR #MA_Cerrar_Centrado) AND #Centrador_EnMovimiento AND NOT #EstadoZona.Manual_CBx,   // "FB910_CNT_UHS"
                  R := NOT #MElev_EnMovimiento,
                  PV := #V_TOut_Centrado,
                  BaseUnidades_ms := "CTE_BaseUnidades_1s");
END_REGION

REGION Network 44: ERROR - TimeOut de Abrir el Centrador
   RUNG wire#powerrail
      Contact( #EstadoZona.Rearme_CBx )
      S_RS(operand := #EstadoMAQ.Err_TimeOut_AbriendoCentrador, s1 := wire#w1)
      S_Coil( #EstadoMAQ.Error_MAQx )
   END_RUNG
   RUNG wire#powerrail
      Contact( #TOut_Centrado.QU )
      Contact( #MA_Abrir_Centrado )
   END_RUNG wire#w1
   // the same network as SCL:
   IF #EstadoZona.Rearme_CBx THEN
       #EstadoMAQ.Err_TimeOut_AbriendoCentrador := FALSE;   // RS flip-flop
   END_IF;
   IF #TOut_Centrado.QU AND #MA_Abrir_Centrado THEN #EstadoMAQ.Err_TimeOut_AbriendoCentrador := TRUE; END_IF;
   IF #EstadoMAQ.Err_TimeOut_AbriendoCentrador THEN #EstadoMAQ.Error_MAQx := TRUE; END_IF;
END_REGION

REGION Network 45: ERROR - TimeOut de Cerrar el Centrador
   RUNG wire#powerrail
      Contact( #EstadoZona.Rearme_CBx )
      S_RS(operand := #EstadoMAQ.Err_TimeOut_CerrandoCentrador, s1 := wire#w1)
      S_Coil( #EstadoMAQ.Error_MAQx )
   END_RUNG
   RUNG wire#powerrail
      Contact( #TOut_Centrado.QU )
      Contact( #MA_Cerrar_Centrado )
   END_RUNG wire#w1
   // the same network as SCL:
   IF #EstadoZona.Rearme_CBx THEN
       #EstadoMAQ.Err_TimeOut_CerrandoCentrador := FALSE;   // RS flip-flop
   END_IF;
   IF #TOut_Centrado.QU AND #MA_Cerrar_Centrado THEN
       #EstadoMAQ.Err_TimeOut_CerrandoCentrador := TRUE;
   END_IF;
   IF #EstadoMAQ.Err_TimeOut_CerrandoCentrador THEN #EstadoMAQ.Error_MAQx := TRUE; END_IF;
END_REGION

REGION Network 46: CONTROL DE TIEMPO - ERROR - Protrusión (Nota: limitacion de Valor a 1 Segundo)
   RUNG wire#powerrail
      Contact( "ON" )
      Move(in := #V_TMP_Protrusion, out1 => #V_Protrusion)
      { S7_Templates := "SrcType := Int" } GT_Contact(in1 := #V_Protrusion, in2 := 1000)
      Move(in := 1000, out1 => #V_Protrusion)
   END_RUNG
   // the same network as SCL:
   IF "ON" THEN #V_Protrusion := #V_TMP_Protrusion; END_IF;
   IF "ON" AND (#V_Protrusion > 1000) THEN #V_Protrusion := 1000; END_IF;
END_REGION

REGION Network 47: TMP - ERROR - Protrusión
   RUNG wire#powerrail
      #TMP_Protrusion(IN := wire#w1, R := wire#w2, PV := #V_Protrusion, BaseUnidades_ms := "CTE_BaseUnidades_1ms", QU =>, QD =>, CVU =>, CVD =>)
   END_RUNG
   RUNG wire#powerrail
      I_Contact( #EstadoVI.Etapas_Carga_E1 )
      I_Contact( #EstadoVI.Etapas_Descarga_S1 )
      I_Contact( #pHsMx_PR1 )
      I_Contact( #Anular_prE1 )
   END_RUNG wire#w1
   RUNG wire#powerrail
      I_Contact( #pHsMx_PR1 )
      I_Contact( #Anular_prE1 )
      Contact( #EstadoZona.Manual_CBx )
   END_RUNG wire#w1
   RUNG wire#powerrail
      Contact( #pHsMx_PR1 )
   END_RUNG wire#w2
   // the same network as SCL:
   #TMP_Protrusion(IN := (NOT #EstadoVI.Etapas_Carga_E1 AND NOT #EstadoVI.Etapas_Descarga_S1 AND NOT #pHsMx_PR1 AND NOT #Anular_prE1) OR (NOT #pHsMx_PR1 AND NOT #Anular_prE1 AND #EstadoZona.Manual_CBx),   // "FB910_CNT_UHS"
                   R := #pHsMx_PR1,
                   PV := #V_Protrusion,
                   BaseUnidades_ms := "CTE_BaseUnidades_1ms");
END_REGION

REGION Network 48: ERROR - Protrusión
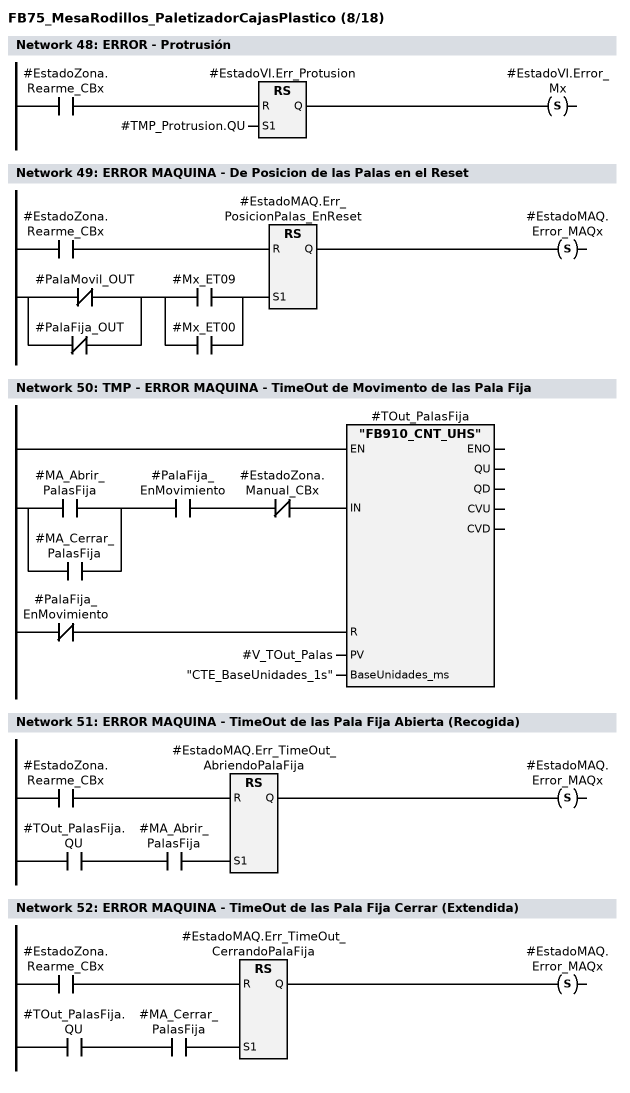
   RUNG wire#powerrail
      Contact( #EstadoZona.Rearme_CBx )
      S_RS(operand := #EstadoVI.Err_Protusion, s1 := #TMP_Protrusion.QU)
      S_Coil( #EstadoVI.Error_Mx )
   END_RUNG
   // the same network as SCL:
   IF #EstadoZona.Rearme_CBx THEN
       #EstadoVI.Err_Protusion := FALSE;   // RS flip-flop
   END_IF;
   IF #TMP_Protrusion.QU THEN #EstadoVI.Err_Protusion := TRUE; END_IF;
   IF #EstadoVI.Err_Protusion THEN #EstadoVI.Error_Mx := TRUE; END_IF;
END_REGION

REGION Network 49: ERROR MAQUINA - De Posicion de las Palas en el Reset
   RUNG wire#powerrail
      Contact( #EstadoZona.Rearme_CBx )
      S_RS(operand := #EstadoMAQ.Err_PosicionPalas_EnReset, s1 := wire#w2)
      S_Coil( #EstadoMAQ.Error_MAQx )
   END_RUNG
   RUNG wire#powerrail
      I_Contact( #PalaMovil_OUT )
      wire#w1
      Contact( #Mx_ET09 )
   END_RUNG wire#w2
   RUNG wire#powerrail
      I_Contact( #PalaFija_OUT )
   END_RUNG wire#w1
   RUNG wire#w1
      Contact( #Mx_ET00 )
   END_RUNG wire#w2
   // the same network as SCL:
   IF #EstadoZona.Rearme_CBx THEN
       #EstadoMAQ.Err_PosicionPalas_EnReset := FALSE;   // RS flip-flop
   END_IF;
   IF (NOT #PalaMovil_OUT OR NOT #PalaFija_OUT) AND (#Mx_ET09 OR #Mx_ET00) THEN
       #EstadoMAQ.Err_PosicionPalas_EnReset := TRUE;
   END_IF;
   IF #EstadoMAQ.Err_PosicionPalas_EnReset THEN #EstadoMAQ.Error_MAQx := TRUE; END_IF;
END_REGION

REGION Network 50: TMP - ERROR MAQUINA - TimeOut de Movimento de las Pala Fija
   RUNG wire#powerrail
      #TOut_PalasFija(IN := wire#w2, R := wire#w3, PV := #V_TOut_Palas, BaseUnidades_ms := "CTE_BaseUnidades_1s", QU =>, QD =>, CVU =>, CVD =>)
   END_RUNG
   RUNG wire#powerrail
      Contact( #MA_Abrir_PalasFija )
      wire#w1
      Contact( #PalaFija_EnMovimiento )
      I_Contact( #EstadoZona.Manual_CBx )
   END_RUNG wire#w2
   RUNG wire#powerrail
      Contact( #MA_Cerrar_PalasFija )
   END_RUNG wire#w1
   RUNG wire#powerrail
      I_Contact( #PalaFija_EnMovimiento )
   END_RUNG wire#w3
   // the same network as SCL:
   #TOut_PalasFija(IN := (#MA_Abrir_PalasFija OR #MA_Cerrar_PalasFija) AND #PalaFija_EnMovimiento AND NOT #EstadoZona.Manual_CBx,   // "FB910_CNT_UHS"
                   R := NOT #PalaFija_EnMovimiento,
                   PV := #V_TOut_Palas,
                   BaseUnidades_ms := "CTE_BaseUnidades_1s");
END_REGION

REGION Network 51: ERROR MAQUINA - TimeOut de las Pala Fija Abierta (Recogida)
   RUNG wire#powerrail
      Contact( #EstadoZona.Rearme_CBx )
      S_RS(operand := #EstadoMAQ.Err_TimeOut_AbriendoPalaFija, s1 := wire#w1)
      S_Coil( #EstadoMAQ.Error_MAQx )
   END_RUNG
   RUNG wire#powerrail
      Contact( #TOut_PalasFija.QU )
      Contact( #MA_Abrir_PalasFija )
   END_RUNG wire#w1
   // the same network as SCL:
   IF #EstadoZona.Rearme_CBx THEN
       #EstadoMAQ.Err_TimeOut_AbriendoPalaFija := FALSE;   // RS flip-flop
   END_IF;
   IF #TOut_PalasFija.QU AND #MA_Abrir_PalasFija THEN
       #EstadoMAQ.Err_TimeOut_AbriendoPalaFija := TRUE;
   END_IF;
   IF #EstadoMAQ.Err_TimeOut_AbriendoPalaFija THEN #EstadoMAQ.Error_MAQx := TRUE; END_IF;
END_REGION

REGION Network 52: ERROR MAQUINA - TimeOut de las Pala Fija Cerrar (Extendida)
   RUNG wire#powerrail
      Contact( #EstadoZona.Rearme_CBx )
      S_RS(operand := #EstadoMAQ.Err_TimeOut_CerrandoPalaFija, s1 := wire#w1)
      S_Coil( #EstadoMAQ.Error_MAQx )
   END_RUNG
   RUNG wire#powerrail
      Contact( #TOut_PalasFija.QU )
      Contact( #MA_Cerrar_PalasFija )
   END_RUNG wire#w1
   // the same network as SCL:
   IF #EstadoZona.Rearme_CBx THEN
       #EstadoMAQ.Err_TimeOut_CerrandoPalaFija := FALSE;   // RS flip-flop
   END_IF;
   IF #TOut_PalasFija.QU AND #MA_Cerrar_PalasFija THEN
       #EstadoMAQ.Err_TimeOut_CerrandoPalaFija := TRUE;
   END_IF;
   IF #EstadoMAQ.Err_TimeOut_CerrandoPalaFija THEN #EstadoMAQ.Error_MAQx := TRUE; END_IF;
END_REGION

REGION Network 53: TMP - ERROR MAQUINA - TimeOut de Movimiento de las Pala Movil
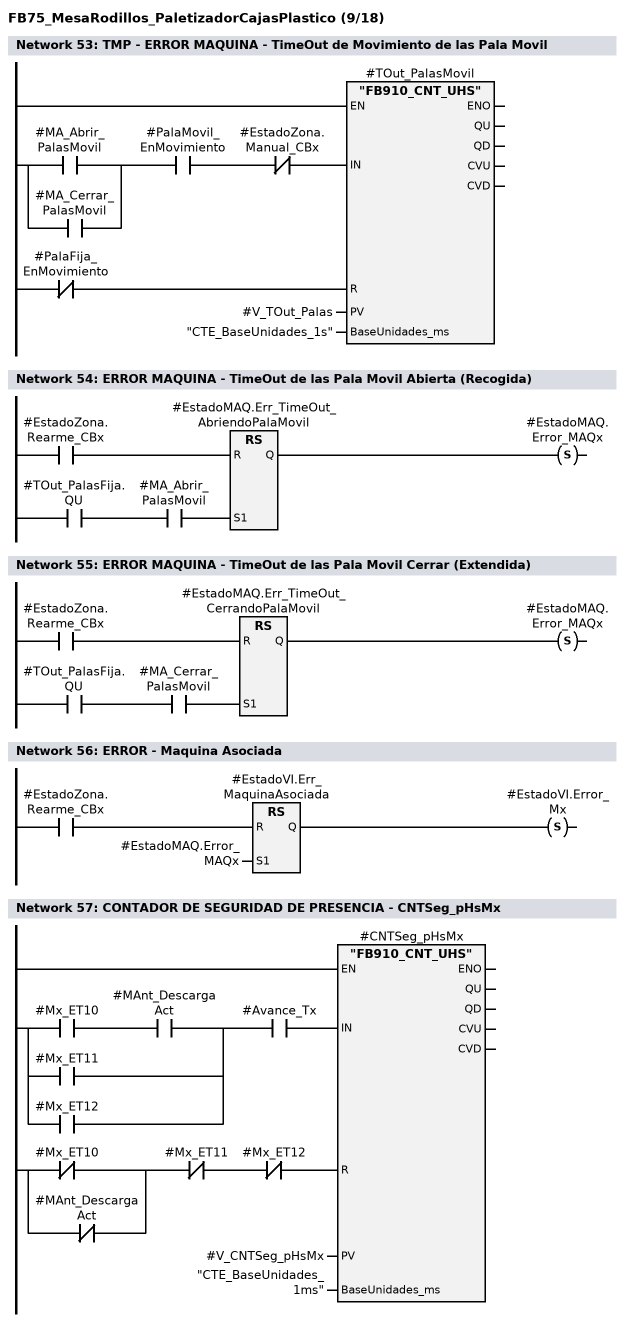
   RUNG wire#powerrail
      #TOut_PalasMovil(IN := wire#w2, R := wire#w3, PV := #V_TOut_Palas, BaseUnidades_ms := "CTE_BaseUnidades_1s", QU =>, QD =>, CVU =>, CVD =>)
   END_RUNG
   RUNG wire#powerrail
      Contact( #MA_Abrir_PalasMovil )
      wire#w1
      Contact( #PalaMovil_EnMovimiento )
      I_Contact( #EstadoZona.Manual_CBx )
   END_RUNG wire#w2
   RUNG wire#powerrail
      Contact( #MA_Cerrar_PalasMovil )
   END_RUNG wire#w1
   RUNG wire#powerrail
      I_Contact( #PalaFija_EnMovimiento )
   END_RUNG wire#w3
   // the same network as SCL:
   #TOut_PalasMovil(IN := (#MA_Abrir_PalasMovil OR #MA_Cerrar_PalasMovil) AND #PalaMovil_EnMovimiento AND NOT #EstadoZona.Manual_CBx,   // "FB910_CNT_UHS"
                    R := NOT #PalaFija_EnMovimiento,
                    PV := #V_TOut_Palas,
                    BaseUnidades_ms := "CTE_BaseUnidades_1s");
END_REGION

REGION Network 54: ERROR MAQUINA - TimeOut de las Pala Movil Abierta (Recogida)
   RUNG wire#powerrail
      Contact( #EstadoZona.Rearme_CBx )
      S_RS(operand := #EstadoMAQ.Err_TimeOut_AbriendoPalaMovil, s1 := wire#w1)
      S_Coil( #EstadoMAQ.Error_MAQx )
   END_RUNG
   RUNG wire#powerrail
      Contact( #TOut_PalasFija.QU )
      Contact( #MA_Abrir_PalasMovil )
   END_RUNG wire#w1
   // the same network as SCL:
   IF #EstadoZona.Rearme_CBx THEN
       #EstadoMAQ.Err_TimeOut_AbriendoPalaMovil := FALSE;   // RS flip-flop
   END_IF;
   IF #TOut_PalasFija.QU AND #MA_Abrir_PalasMovil THEN
       #EstadoMAQ.Err_TimeOut_AbriendoPalaMovil := TRUE;
   END_IF;
   IF #EstadoMAQ.Err_TimeOut_AbriendoPalaMovil THEN #EstadoMAQ.Error_MAQx := TRUE; END_IF;
END_REGION

REGION Network 55: ERROR MAQUINA - TimeOut de las Pala Movil Cerrar (Extendida)
   RUNG wire#powerrail
      Contact( #EstadoZona.Rearme_CBx )
      S_RS(operand := #EstadoMAQ.Err_TimeOut_CerrandoPalaMovil, s1 := wire#w1)
      S_Coil( #EstadoMAQ.Error_MAQx )
   END_RUNG
   RUNG wire#powerrail
      Contact( #TOut_PalasFija.QU )
      Contact( #MA_Cerrar_PalasMovil )
   END_RUNG wire#w1
   // the same network as SCL:
   IF #EstadoZona.Rearme_CBx THEN
       #EstadoMAQ.Err_TimeOut_CerrandoPalaMovil := FALSE;   // RS flip-flop
   END_IF;
   IF #TOut_PalasFija.QU AND #MA_Cerrar_PalasMovil THEN
       #EstadoMAQ.Err_TimeOut_CerrandoPalaMovil := TRUE;
   END_IF;
   IF #EstadoMAQ.Err_TimeOut_CerrandoPalaMovil THEN #EstadoMAQ.Error_MAQx := TRUE; END_IF;
END_REGION

REGION Network 56: ERROR - Maquina Asociada
   RUNG wire#powerrail
      Contact( #EstadoZona.Rearme_CBx )
      S_RS(operand := #EstadoVI.Err_MaquinaAsociada, s1 := #EstadoMAQ.Error_MAQx)
      S_Coil( #EstadoVI.Error_Mx )
   END_RUNG
   // the same network as SCL:
   IF #EstadoZona.Rearme_CBx THEN
       #EstadoVI.Err_MaquinaAsociada := FALSE;   // RS flip-flop
   END_IF;
   IF #EstadoMAQ.Error_MAQx THEN #EstadoVI.Err_MaquinaAsociada := TRUE; END_IF;
   IF #EstadoVI.Err_MaquinaAsociada THEN #EstadoVI.Error_Mx := TRUE; END_IF;
END_REGION

REGION Network 57: CONTADOR DE SEGURIDAD DE PRESENCIA - CNTSeg_pHsMx
   RUNG wire#powerrail
      #CNTSeg_pHsMx(IN := wire#w2, R := wire#w4, PV := #V_CNTSeg_pHsMx, BaseUnidades_ms := "CTE_BaseUnidades_1ms", QU =>, QD =>, CVU =>, CVD =>)
   END_RUNG
   RUNG wire#powerrail
      Contact( #Mx_ET10 )
      Contact( #MAnt_DescargaAct )
      wire#w1
      Contact( #Avance_Tx )
   END_RUNG wire#w2
   RUNG wire#powerrail
      Contact( #Mx_ET11 )
   END_RUNG wire#w1
   RUNG wire#powerrail
      Contact( #Mx_ET12 )
   END_RUNG wire#w1
   RUNG wire#powerrail
      I_Contact( #Mx_ET10 )
      wire#w3
      I_Contact( #Mx_ET11 )
      I_Contact( #Mx_ET12 )
   END_RUNG wire#w4
   RUNG wire#powerrail
      I_Contact( #MAnt_DescargaAct )
   END_RUNG wire#w3
   // the same network as SCL:
   #CNTSeg_pHsMx(IN := ((#Mx_ET10 AND #MAnt_DescargaAct) OR #Mx_ET11 OR #Mx_ET12) AND #Avance_Tx,   // "FB910_CNT_UHS"
                 R := (NOT #Mx_ET10 OR NOT #MAnt_DescargaAct) AND NOT #Mx_ET11 AND NOT #Mx_ET12,
                 PV := #V_CNTSeg_pHsMx,
                 BaseUnidades_ms := "CTE_BaseUnidades_1ms");
END_REGION

REGION Network 58: CONTADOR DE PRESENCIA - CNT_pHsMx
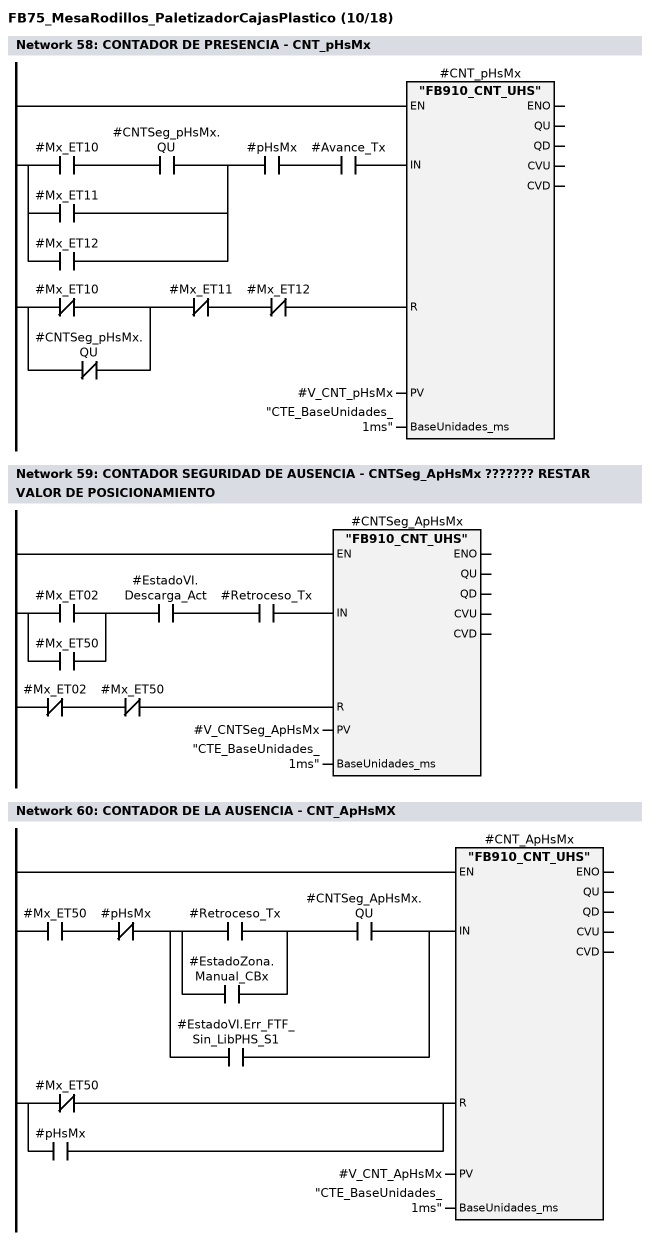
   RUNG wire#powerrail
      #CNT_pHsMx(IN := wire#w2, R := wire#w4, PV := #V_CNT_pHsMx, BaseUnidades_ms := "CTE_BaseUnidades_1ms", QU =>, QD =>, CVU =>, CVD =>)
   END_RUNG
   RUNG wire#powerrail
      Contact( #Mx_ET10 )
      Contact( #CNTSeg_pHsMx.QU )
      wire#w1
      Contact( #pHsMx )
      Contact( #Avance_Tx )
   END_RUNG wire#w2
   RUNG wire#powerrail
      Contact( #Mx_ET11 )
   END_RUNG wire#w1
   RUNG wire#powerrail
      Contact( #Mx_ET12 )
   END_RUNG wire#w1
   RUNG wire#powerrail
      I_Contact( #Mx_ET10 )
      wire#w3
      I_Contact( #Mx_ET11 )
      I_Contact( #Mx_ET12 )
   END_RUNG wire#w4
   RUNG wire#powerrail
      I_Contact( #CNTSeg_pHsMx.QU )
   END_RUNG wire#w3
   // the same network as SCL:
   #CNT_pHsMx(IN := ((#Mx_ET10 AND #CNTSeg_pHsMx.QU) OR #Mx_ET11 OR #Mx_ET12) AND #pHsMx AND #Avance_Tx,   // "FB910_CNT_UHS"
              R := (NOT #Mx_ET10 OR NOT #CNTSeg_pHsMx.QU) AND NOT #Mx_ET11 AND NOT #Mx_ET12,
              PV := #V_CNT_pHsMx,
              BaseUnidades_ms := "CTE_BaseUnidades_1ms");
END_REGION

REGION Network 59: CONTADOR SEGURIDAD DE AUSENCIA - CNTSeg_ApHsMx ??????? RESTAR VALOR DE POSICIONAMIENTO
   RUNG wire#powerrail
      #CNTSeg_ApHsMx(IN := wire#w2, R := wire#w3, PV := #V_CNTSeg_ApHsMx, BaseUnidades_ms := "CTE_BaseUnidades_1ms", QU =>, QD =>, CVU =>, CVD =>)
   END_RUNG
   RUNG wire#powerrail
      Contact( #Mx_ET02 )
      wire#w1
      Contact( #EstadoVI.Descarga_Act )
      Contact( #Retroceso_Tx )
   END_RUNG wire#w2
   RUNG wire#powerrail
      Contact( #Mx_ET50 )
   END_RUNG wire#w1
   RUNG wire#powerrail
      I_Contact( #Mx_ET02 )
      I_Contact( #Mx_ET50 )
   END_RUNG wire#w3
   // the same network as SCL:
   #CNTSeg_ApHsMx(IN := (#Mx_ET02 OR #Mx_ET50) AND #EstadoVI.Descarga_Act AND #Retroceso_Tx,   // "FB910_CNT_UHS"
                  R := NOT #Mx_ET02 AND NOT #Mx_ET50,
                  PV := #V_CNTSeg_ApHsMx,
                  BaseUnidades_ms := "CTE_BaseUnidades_1ms");
END_REGION

REGION Network 60: CONTADOR DE LA AUSENCIA - CNT_ApHsMX
   RUNG wire#powerrail
      #CNT_ApHsMx(IN := wire#w3, R := wire#w4, PV := #V_CNT_ApHsMx, BaseUnidades_ms := "CTE_BaseUnidades_1ms", QU =>, QD =>, CVU =>, CVD =>)
   END_RUNG
   RUNG wire#powerrail
      Contact( #Mx_ET50 )
      I_Contact( #pHsMx )
      wire#w1
      Contact( #Retroceso_Tx )
      wire#w2
      Contact( #CNTSeg_ApHsMx.QU )
   END_RUNG wire#w3
   RUNG wire#w1
      Contact( #EstadoZona.Manual_CBx )
   END_RUNG wire#w2
   RUNG wire#w1
      Contact( #EstadoVI.Err_FTF_Sin_LibPHS_S1 )
   END_RUNG wire#w3
   RUNG wire#powerrail
      I_Contact( #Mx_ET50 )
   END_RUNG wire#w4
   RUNG wire#powerrail
      Contact( #pHsMx )
   END_RUNG wire#w4
   // the same network as SCL:
   #CNT_ApHsMx(IN := #Mx_ET50 AND NOT #pHsMx AND (((#Retroceso_Tx OR #EstadoZona.Manual_CBx) AND #CNTSeg_ApHsMx.QU) OR #EstadoVI.Err_FTF_Sin_LibPHS_S1),   // "FB910_CNT_UHS"
               R := NOT #Mx_ET50 OR #pHsMx,
               PV := #V_CNT_ApHsMx,
               BaseUnidades_ms := "CTE_BaseUnidades_1ms");
END_REGION

REGION Network 61: TEMPORIZADOR DE ESTABILIDAD DE LA PALA MOVIL
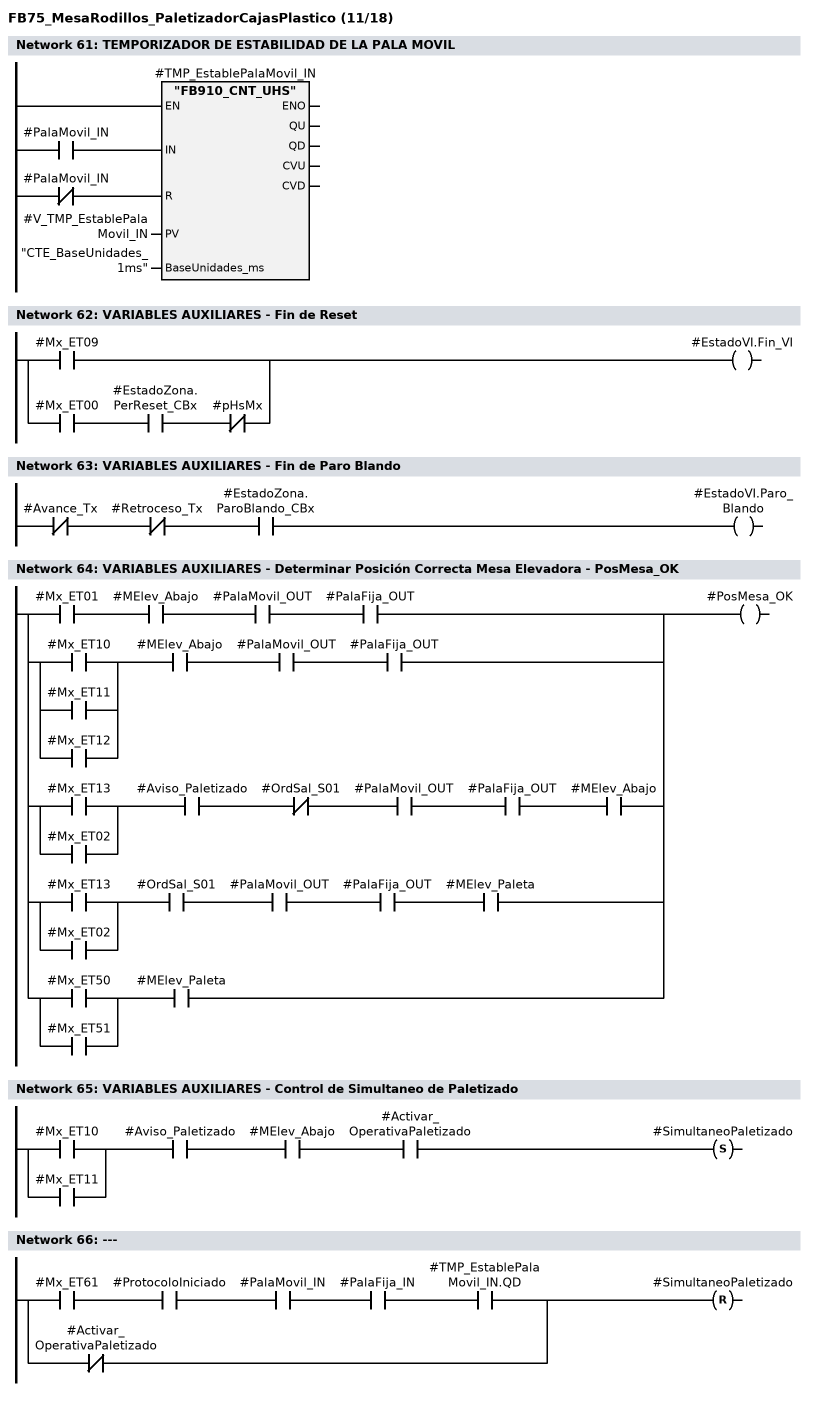
   RUNG wire#powerrail
      #TMP_EstablePalaMovil_IN(IN := wire#w1, R := wire#w2, PV := #V_TMP_EstablePalaMovil_IN, BaseUnidades_ms := "CTE_BaseUnidades_1ms", QU =>, QD =>, CVU =>, CVD =>)
   END_RUNG
   RUNG wire#powerrail
      Contact( #PalaMovil_IN )
   END_RUNG wire#w1
   RUNG wire#powerrail
      I_Contact( #PalaMovil_IN )
   END_RUNG wire#w2
   // the same network as SCL:
   #TMP_EstablePalaMovil_IN(IN := #PalaMovil_IN,   // "FB910_CNT_UHS"
                           R := NOT #PalaMovil_IN,
                           PV := #V_TMP_EstablePalaMovil_IN,
                           BaseUnidades_ms := "CTE_BaseUnidades_1ms");
END_REGION

REGION Network 62: VARIABLES AUXILIARES - Fin de Reset
   RUNG wire#powerrail
      Contact( #Mx_ET09 )
      wire#w1
      Coil( #EstadoVI.Fin_VI )
   END_RUNG
   RUNG wire#powerrail
      Contact( #Mx_ET00 )
      Contact( #EstadoZona.PerReset_CBx )
      I_Contact( #pHsMx )
   END_RUNG wire#w1
   // the same network as SCL:
   #EstadoVI.Fin_VI := #Mx_ET09 OR (#Mx_ET00 AND #EstadoZona.PerReset_CBx AND NOT #pHsMx);
END_REGION

REGION Network 63: VARIABLES AUXILIARES - Fin de Paro Blando
   RUNG wire#powerrail
      I_Contact( #Avance_Tx )
      I_Contact( #Retroceso_Tx )
      Contact( #EstadoZona.ParoBlando_CBx )
      Coil( #EstadoVI.Paro_Blando )
   END_RUNG
   // the same network as SCL:
   #EstadoVI.Paro_Blando := NOT #Avance_Tx AND NOT #Retroceso_Tx AND #EstadoZona.ParoBlando_CBx;
END_REGION

REGION Network 64: VARIABLES AUXILIARES - Determinar Posición Correcta Mesa Elevadora - PosMesa_OK
   RUNG wire#powerrail
      Contact( #Mx_ET01 )
      Contact( #MElev_Abajo )
      Contact( #PalaMovil_OUT )
      Contact( #PalaFija_OUT )
      wire#w1
      Coil( #PosMesa_OK )
   END_RUNG
   RUNG wire#powerrail
      Contact( #Mx_ET10 )
      wire#w2
      Contact( #MElev_Abajo )
      Contact( #PalaMovil_OUT )
      Contact( #PalaFija_OUT )
   END_RUNG wire#w1
   RUNG wire#powerrail
      Contact( #Mx_ET11 )
   END_RUNG wire#w2
   RUNG wire#powerrail
      Contact( #Mx_ET12 )
   END_RUNG wire#w2
   RUNG wire#powerrail
      Contact( #Mx_ET13 )
      wire#w3
      Contact( #Aviso_Paletizado )
      I_Contact( #OrdSal_S01 )
      Contact( #PalaMovil_OUT )
      Contact( #PalaFija_OUT )
      Contact( #MElev_Abajo )
   END_RUNG wire#w1
   RUNG wire#powerrail
      Contact( #Mx_ET02 )
   END_RUNG wire#w3
   RUNG wire#powerrail
      Contact( #Mx_ET13 )
      wire#w4
      Contact( #OrdSal_S01 )
      Contact( #PalaMovil_OUT )
      Contact( #PalaFija_OUT )
      Contact( #MElev_Paleta )
   END_RUNG wire#w1
   RUNG wire#powerrail
      Contact( #Mx_ET02 )
   END_RUNG wire#w4
   RUNG wire#powerrail
      Contact( #Mx_ET50 )
      wire#w5
      Contact( #MElev_Paleta )
   END_RUNG wire#w1
   RUNG wire#powerrail
      Contact( #Mx_ET51 )
   END_RUNG wire#w5
   // the same network as SCL:
   #PosMesa_OK := (#Mx_ET01 AND #MElev_Abajo AND #PalaMovil_OUT AND #PalaFija_OUT) OR ((#Mx_ET10 OR #Mx_ET11 OR #Mx_ET12) AND #MElev_Abajo AND #PalaMovil_OUT AND #PalaFija_OUT) OR ((#Mx_ET13 OR #Mx_ET02) AND #Aviso_Paletizado AND NOT #OrdSal_S01 AND #PalaMovil_OUT AND #PalaFija_OUT AND #MElev_Abajo) OR ((#Mx_ET13 OR #Mx_ET02) AND #OrdSal_S01 AND #PalaMovil_OUT AND #PalaFija_OUT AND #MElev_Paleta) OR ((#Mx_ET50 OR #Mx_ET51) AND #MElev_Paleta);
END_REGION

REGION Network 65: VARIABLES AUXILIARES - Control de Simultaneo de Paletizado
   RUNG wire#powerrail
      Contact( #Mx_ET10 )
      wire#w1
      Contact( #Aviso_Paletizado )
      Contact( #MElev_Abajo )
      Contact( #Activar_OperativaPaletizado )
      S_Coil( #SimultaneoPaletizado )
   END_RUNG
   RUNG wire#powerrail
      Contact( #Mx_ET11 )
   END_RUNG wire#w1
   // the same network as SCL:
   IF (#Mx_ET10 OR #Mx_ET11) AND #Aviso_Paletizado AND #MElev_Abajo AND #Activar_OperativaPaletizado THEN
       #SimultaneoPaletizado := TRUE;
   END_IF;
END_REGION

REGION Network 66: ---
   RUNG wire#powerrail
      Contact( #Mx_ET61 )
      Contact( #ProtocoloIniciado )
      Contact( #PalaMovil_IN )
      Contact( #PalaFija_IN )
      Contact( #TMP_EstablePalaMovil_IN.QD )
      wire#w1
      R_Coil( #SimultaneoPaletizado )
   END_RUNG
   RUNG wire#powerrail
      I_Contact( #Activar_OperativaPaletizado )
   END_RUNG wire#w1
   // the same network as SCL:
   IF (#Mx_ET61 AND #ProtocoloIniciado AND #PalaMovil_IN AND #PalaFija_IN AND #TMP_EstablePalaMovil_IN.QD) OR NOT #Activar_OperativaPaletizado THEN
       #SimultaneoPaletizado := FALSE;
   END_IF;
END_REGION

REGION Network 67: VARIABLES AUXILIARES - Permiso de Entrada - PTF_MAnt_Mx
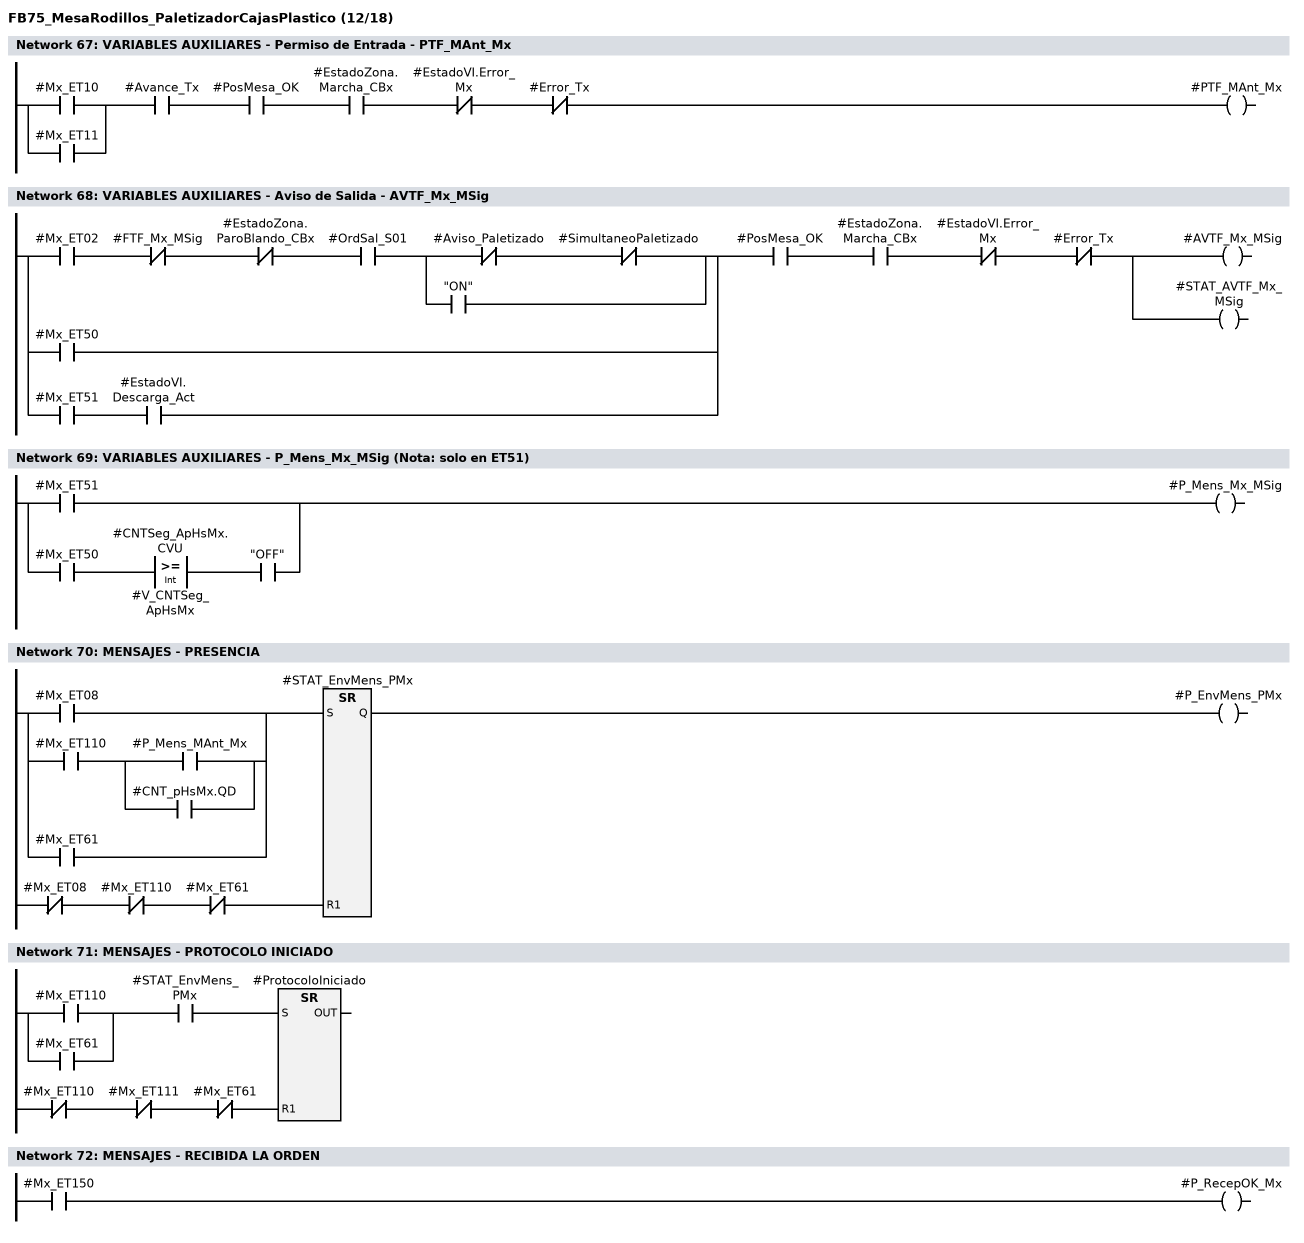
   RUNG wire#powerrail
      Contact( #Mx_ET10 )
      wire#w1
      Contact( #Avance_Tx )
      Contact( #PosMesa_OK )
      Contact( #EstadoZona.Marcha_CBx )
      I_Contact( #EstadoVI.Error_Mx )
      I_Contact( #Error_Tx )
      Coil( #PTF_MAnt_Mx )
   END_RUNG
   RUNG wire#powerrail
      Contact( #Mx_ET11 )
   END_RUNG wire#w1
   // the same network as SCL:
   #PTF_MAnt_Mx := (#Mx_ET10 OR #Mx_ET11) AND #Avance_Tx AND #PosMesa_OK AND #EstadoZona.Marcha_CBx AND NOT #EstadoVI.Error_Mx AND NOT #Error_Tx;
END_REGION

REGION Network 68: VARIABLES AUXILIARES - Aviso de Salida - AVTF_Mx_MSig
   RUNG wire#powerrail
      Contact( #Mx_ET02 )
      I_Contact( #FTF_Mx_MSig )
      I_Contact( #EstadoZona.ParoBlando_CBx )
      Contact( #OrdSal_S01 )
      wire#w1
      I_Contact( #Aviso_Paletizado )
      I_Contact( #SimultaneoPaletizado )
      wire#w2
      Contact( #PosMesa_OK )
      Contact( #EstadoZona.Marcha_CBx )
      I_Contact( #EstadoVI.Error_Mx )
      I_Contact( #Error_Tx )
      wire#w3
      Coil( #AVTF_Mx_MSig )
   END_RUNG
   RUNG wire#w1
      Contact( "ON" )
   END_RUNG wire#w2
   RUNG wire#powerrail
      Contact( #Mx_ET50 )
   END_RUNG wire#w2
   RUNG wire#powerrail
      Contact( #Mx_ET51 )
      Contact( #EstadoVI.Descarga_Act )
   END_RUNG wire#w2
   RUNG wire#w3
      Coil( #STAT_AVTF_Mx_MSig )
   END_RUNG
   // the same network as SCL:
   #AVTF_Mx_MSig := ((#Mx_ET02 AND NOT #FTF_Mx_MSig AND NOT #EstadoZona.ParoBlando_CBx AND #OrdSal_S01 AND ((NOT #Aviso_Paletizado AND NOT #SimultaneoPaletizado) OR "ON")) OR #Mx_ET50 OR (#Mx_ET51 AND #EstadoVI.Descarga_Act)) AND #PosMesa_OK AND #EstadoZona.Marcha_CBx AND NOT #EstadoVI.Error_Mx AND NOT #Error_Tx;
   #STAT_AVTF_Mx_MSig := #AVTF_Mx_MSig;
END_REGION

REGION Network 69: VARIABLES AUXILIARES - P_Mens_Mx_MSig (Nota: solo en ET51)
   RUNG wire#powerrail
      Contact( #Mx_ET51 )
      wire#w1
      Coil( #P_Mens_Mx_MSig )
   END_RUNG
   RUNG wire#powerrail
      Contact( #Mx_ET50 )
      { S7_Templates := "SrcType := Int" } GE_Contact(in1 := #CNTSeg_ApHsMx.CVU, in2 := #V_CNTSeg_ApHsMx)
      Contact( "OFF" )
   END_RUNG wire#w1
   // the same network as SCL:
   #P_Mens_Mx_MSig := #Mx_ET51 OR (#Mx_ET50 AND (#CNTSeg_ApHsMx.CVU >= #V_CNTSeg_ApHsMx) AND "OFF");
END_REGION

REGION Network 70: MENSAJES - PRESENCIA
   RUNG wire#powerrail
      Contact( #Mx_ET08 )
      wire#w1
      S_SR(operand := #STAT_EnvMens_PMx, r1 := wire#w3)
      Coil( #P_EnvMens_PMx )
   END_RUNG
   RUNG wire#powerrail
      Contact( #Mx_ET110 )
      wire#w2
      Contact( #P_Mens_MAnt_Mx )
   END_RUNG wire#w1
   RUNG wire#w2
      Contact( #CNT_pHsMx.QD )
   END_RUNG wire#w1
   RUNG wire#powerrail
      Contact( #Mx_ET61 )
   END_RUNG wire#w1
   RUNG wire#powerrail
      I_Contact( #Mx_ET08 )
      I_Contact( #Mx_ET110 )
      I_Contact( #Mx_ET61 )
   END_RUNG wire#w3
   // the same network as SCL:
   IF #Mx_ET08 OR (#Mx_ET110 AND (#P_Mens_MAnt_Mx OR #CNT_pHsMx.QD)) OR #Mx_ET61 THEN
       #STAT_EnvMens_PMx := TRUE;   // SR flip-flop
   END_IF;
   IF NOT #Mx_ET08 AND NOT #Mx_ET110 AND NOT #Mx_ET61 THEN #STAT_EnvMens_PMx := FALSE; END_IF;
   #P_EnvMens_PMx := #STAT_EnvMens_PMx;
END_REGION

REGION Network 71: MENSAJES - PROTOCOLO INICIADO
   RUNG wire#powerrail
      Contact( #Mx_ET110 )
      wire#w1
      Contact( #STAT_EnvMens_PMx )
      S_SR(operand := #ProtocoloIniciado, r1 := wire#w2)
   END_RUNG
   RUNG wire#powerrail
      Contact( #Mx_ET61 )
   END_RUNG wire#w1
   RUNG wire#powerrail
      I_Contact( #Mx_ET110 )
      I_Contact( #Mx_ET111 )
      I_Contact( #Mx_ET61 )
   END_RUNG wire#w2
   // the same network as SCL:
   IF (#Mx_ET110 OR #Mx_ET61) AND #STAT_EnvMens_PMx THEN
       #ProtocoloIniciado := TRUE;   // SR flip-flop
   END_IF;
   IF NOT #Mx_ET110 AND NOT #Mx_ET111 AND NOT #Mx_ET61 THEN #ProtocoloIniciado := FALSE; END_IF;
END_REGION

REGION Network 72: MENSAJES - RECIBIDA LA ORDEN
   RUNG wire#powerrail
      Contact( #Mx_ET150 )
      Coil( #P_RecepOK_Mx )
   END_RUNG
   // the same network as SCL:
   #P_RecepOK_Mx := #Mx_ET150;
END_REGION

REGION Network 73: INTERLOCK - Mesa de Banda del Paletizador de Cajas de Plastico
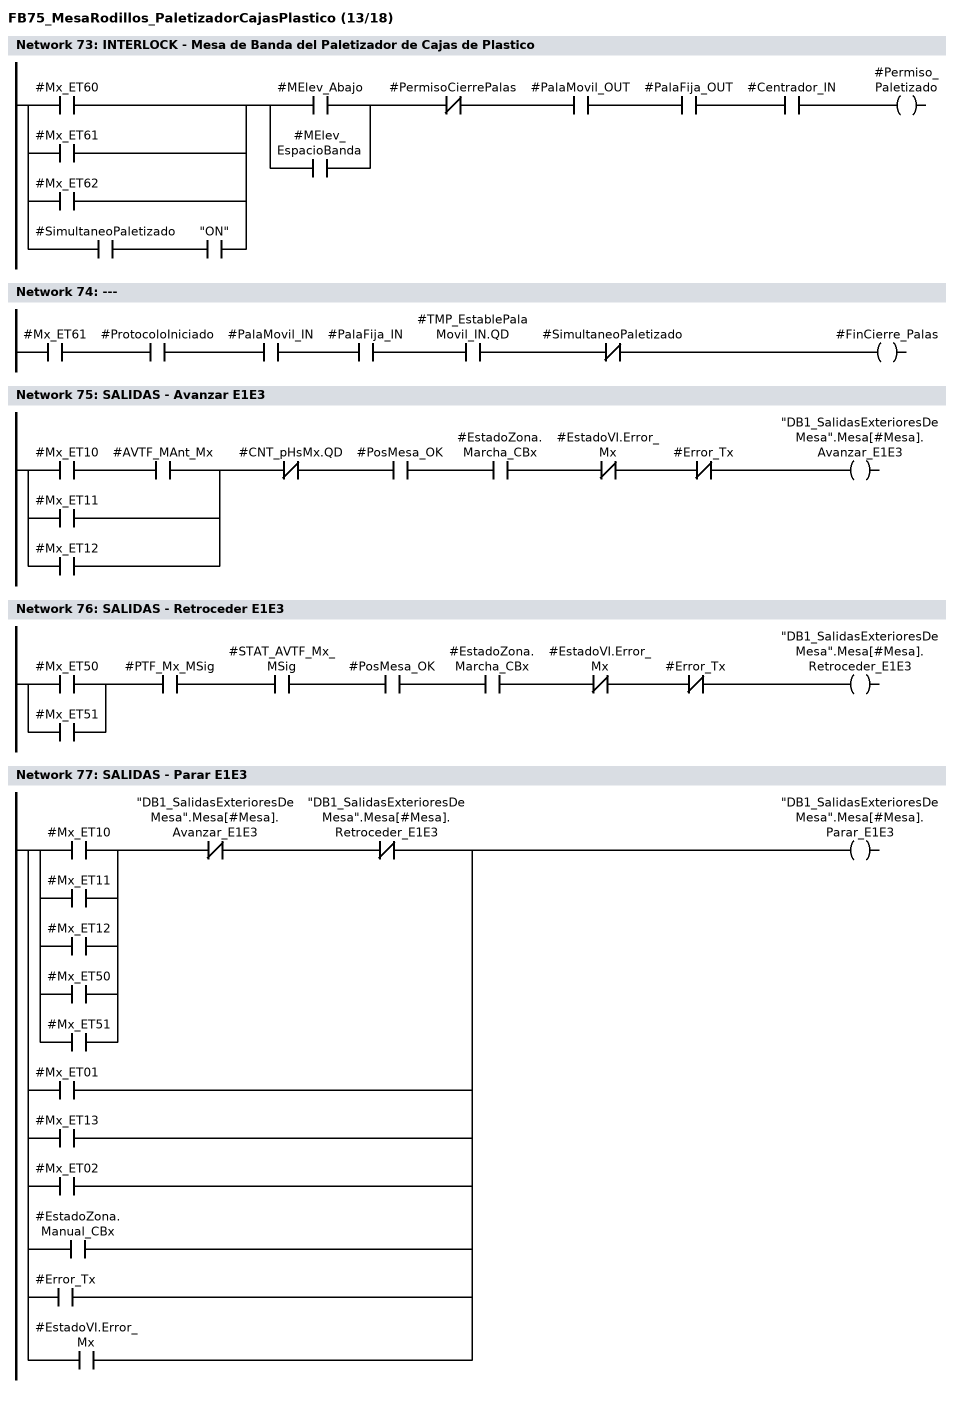
   RUNG wire#powerrail
      Contact( #Mx_ET60 )
      wire#w1
      Contact( #MElev_Abajo )
      wire#w2
      I_Contact( #PermisoCierrePalas )
      Contact( #PalaMovil_OUT )
      Contact( #PalaFija_OUT )
      Contact( #Centrador_IN )
      Coil( #Permiso_Paletizado )
   END_RUNG
   RUNG wire#powerrail
      Contact( #Mx_ET61 )
   END_RUNG wire#w1
   RUNG wire#powerrail
      Contact( #Mx_ET62 )
   END_RUNG wire#w1
   RUNG wire#powerrail
      Contact( #SimultaneoPaletizado )
      Contact( "ON" )
   END_RUNG wire#w1
   RUNG wire#w1
      Contact( #MElev_EspacioBanda )
   END_RUNG wire#w2
   // the same network as SCL:
   #Permiso_Paletizado := (#Mx_ET60 OR #Mx_ET61 OR #Mx_ET62 OR (#SimultaneoPaletizado AND "ON")) AND (#MElev_Abajo OR #MElev_EspacioBanda) AND NOT #PermisoCierrePalas AND #PalaMovil_OUT AND #PalaFija_OUT AND #Centrador_IN;
END_REGION

REGION Network 74: ---
   RUNG wire#powerrail
      Contact( #Mx_ET61 )
      Contact( #ProtocoloIniciado )
      Contact( #PalaMovil_IN )
      Contact( #PalaFija_IN )
      Contact( #TMP_EstablePalaMovil_IN.QD )
      I_Contact( #SimultaneoPaletizado )
      Coil( #FinCierre_Palas )
   END_RUNG
   // the same network as SCL:
   #FinCierre_Palas := #Mx_ET61 AND #ProtocoloIniciado AND #PalaMovil_IN AND #PalaFija_IN AND #TMP_EstablePalaMovil_IN.QD AND NOT #SimultaneoPaletizado;
END_REGION

REGION Network 75: SALIDAS - Avanzar E1E3
   RUNG wire#powerrail
      Contact( #Mx_ET10 )
      Contact( #AVTF_MAnt_Mx )
      wire#w1
      I_Contact( #CNT_pHsMx.QD )
      Contact( #PosMesa_OK )
      Contact( #EstadoZona.Marcha_CBx )
      I_Contact( #EstadoVI.Error_Mx )
      I_Contact( #Error_Tx )
      Coil( "DB1_SalidasExterioresDeMesa".Mesa[#Mesa].Avanzar_E1E3 )
   END_RUNG
   RUNG wire#powerrail
      Contact( #Mx_ET11 )
   END_RUNG wire#w1
   RUNG wire#powerrail
      Contact( #Mx_ET12 )
   END_RUNG wire#w1
   // the same network as SCL:
   "DB1_SalidasExterioresDeMesa".Mesa[#Mesa].Avanzar_E1E3 := ((#Mx_ET10 AND #AVTF_MAnt_Mx) OR #Mx_ET11 OR #Mx_ET12) AND NOT #CNT_pHsMx.QD AND #PosMesa_OK AND #EstadoZona.Marcha_CBx AND NOT #EstadoVI.Error_Mx AND NOT #Error_Tx;
END_REGION

REGION Network 76: SALIDAS - Retroceder E1E3
   RUNG wire#powerrail
      Contact( #Mx_ET50 )
      wire#w1
      Contact( #PTF_Mx_MSig )
      Contact( #STAT_AVTF_Mx_MSig )
      Contact( #PosMesa_OK )
      Contact( #EstadoZona.Marcha_CBx )
      I_Contact( #EstadoVI.Error_Mx )
      I_Contact( #Error_Tx )
      Coil( "DB1_SalidasExterioresDeMesa".Mesa[#Mesa].Retroceder_E1E3 )
   END_RUNG
   RUNG wire#powerrail
      Contact( #Mx_ET51 )
   END_RUNG wire#w1
   // the same network as SCL:
   "DB1_SalidasExterioresDeMesa".Mesa[#Mesa].Retroceder_E1E3 := (#Mx_ET50 OR #Mx_ET51) AND #PTF_Mx_MSig AND #STAT_AVTF_Mx_MSig AND #PosMesa_OK AND #EstadoZona.Marcha_CBx AND NOT #EstadoVI.Error_Mx AND NOT #Error_Tx;
END_REGION

REGION Network 77: SALIDAS - Parar E1E3
   RUNG wire#powerrail
      Contact( #Mx_ET10 )
      wire#w1
      I_Contact( "DB1_SalidasExterioresDeMesa".Mesa[#Mesa].Avanzar_E1E3 )
      I_Contact( "DB1_SalidasExterioresDeMesa".Mesa[#Mesa].Retroceder_E1E3 )
      wire#w2
      Coil( "DB1_SalidasExterioresDeMesa".Mesa[#Mesa].Parar_E1E3 )
   END_RUNG
   RUNG wire#powerrail
      Contact( #Mx_ET11 )
   END_RUNG wire#w1
   RUNG wire#powerrail
      Contact( #Mx_ET12 )
   END_RUNG wire#w1
   RUNG wire#powerrail
      Contact( #Mx_ET50 )
   END_RUNG wire#w1
   RUNG wire#powerrail
      Contact( #Mx_ET51 )
   END_RUNG wire#w1
   RUNG wire#powerrail
      Contact( #Mx_ET01 )
   END_RUNG wire#w2
   RUNG wire#powerrail
      Contact( #Mx_ET13 )
   END_RUNG wire#w2
   RUNG wire#powerrail
      Contact( #Mx_ET02 )
   END_RUNG wire#w2
   RUNG wire#powerrail
      Contact( #EstadoZona.Manual_CBx )
   END_RUNG wire#w2
   RUNG wire#powerrail
      Contact( #Error_Tx )
   END_RUNG wire#w2
   RUNG wire#powerrail
      Contact( #EstadoVI.Error_Mx )
   END_RUNG wire#w2
   // the same network as SCL:
   "DB1_SalidasExterioresDeMesa".Mesa[#Mesa].Parar_E1E3 := ((#Mx_ET10 OR #Mx_ET11 OR #Mx_ET12 OR #Mx_ET50 OR #Mx_ET51) AND NOT "DB1_SalidasExterioresDeMesa".Mesa[#Mesa].Avanzar_E1E3 AND NOT "DB1_SalidasExterioresDeMesa".Mesa[#Mesa].Retroceder_E1E3) OR #Mx_ET01 OR #Mx_ET13 OR #Mx_ET02 OR #EstadoZona.Manual_CBx OR #Error_Tx OR #EstadoVI.Error_Mx;
END_REGION

REGION Network 78: SALIDAS - Valor Frecuencia Lenta E1E3
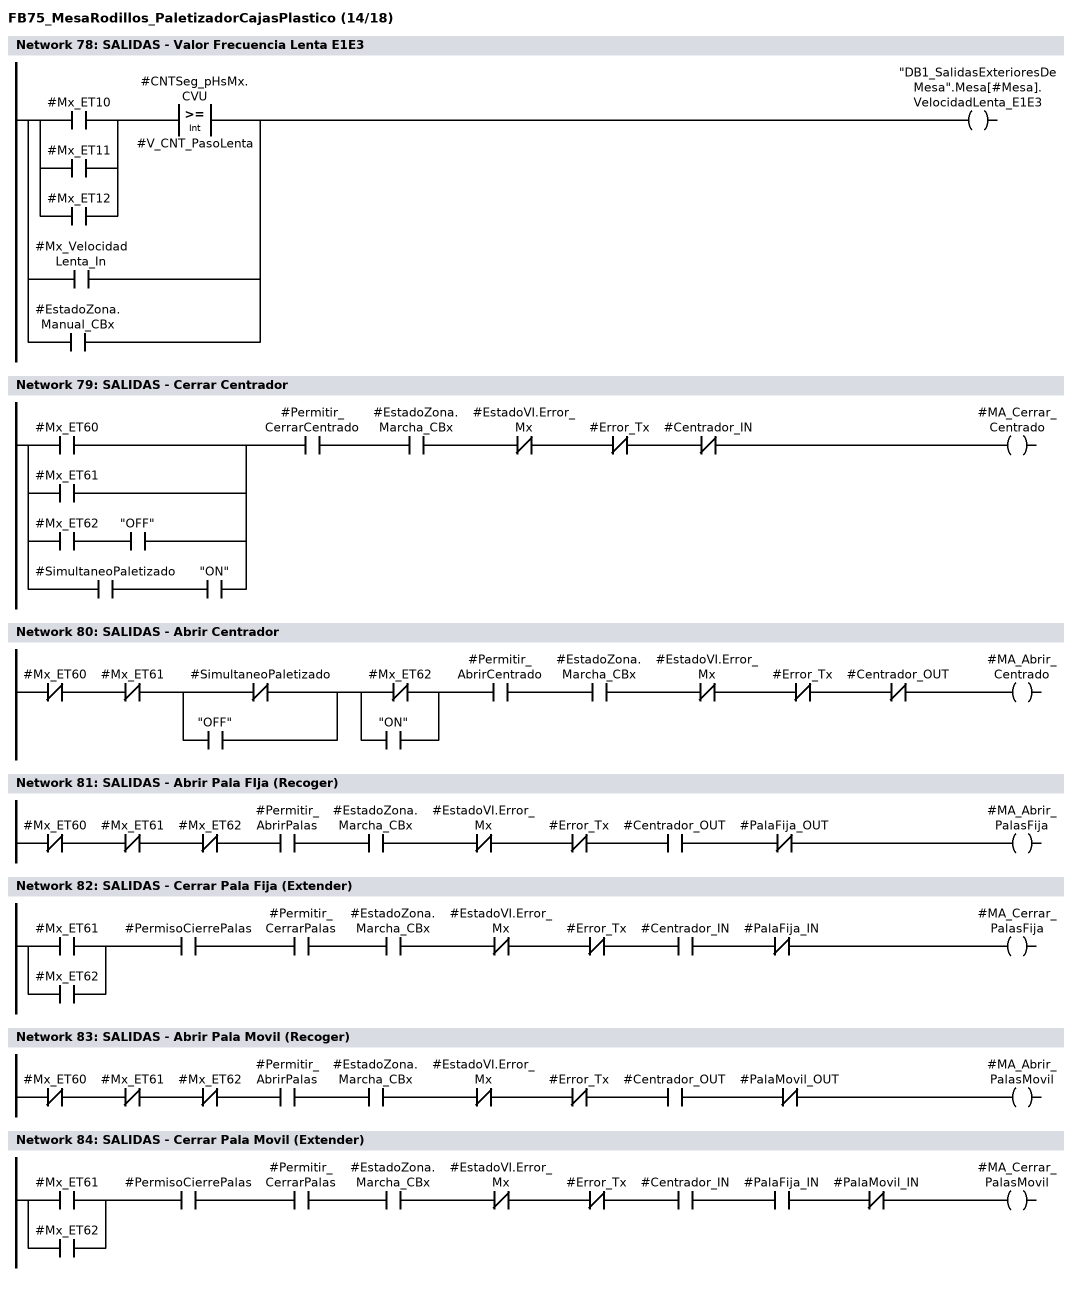
   RUNG wire#powerrail
      Contact( #Mx_ET10 )
      wire#w1
      { S7_Templates := "SrcType := Int" } GE_Contact(in1 := #CNTSeg_pHsMx.CVU, in2 := #V_CNT_PasoLenta)
      wire#w2
      Coil( "DB1_SalidasExterioresDeMesa".Mesa[#Mesa].VelocidadLenta_E1E3 )
   END_RUNG
   RUNG wire#powerrail
      Contact( #Mx_ET11 )
   END_RUNG wire#w1
   RUNG wire#powerrail
      Contact( #Mx_ET12 )
   END_RUNG wire#w1
   RUNG wire#powerrail
      Contact( #Mx_VelocidadLenta_In )
   END_RUNG wire#w2
   RUNG wire#powerrail
      Contact( #EstadoZona.Manual_CBx )
   END_RUNG wire#w2
   // the same network as SCL:
   "DB1_SalidasExterioresDeMesa".Mesa[#Mesa].VelocidadLenta_E1E3 := ((#Mx_ET10 OR #Mx_ET11 OR #Mx_ET12) AND (#CNTSeg_pHsMx.CVU >= #V_CNT_PasoLenta)) OR #Mx_VelocidadLenta_In OR #EstadoZona.Manual_CBx;
END_REGION

REGION Network 79: SALIDAS - Cerrar Centrador
   RUNG wire#powerrail
      Contact( #Mx_ET60 )
      wire#w1
      Contact( #Permitir_CerrarCentrado )
      Contact( #EstadoZona.Marcha_CBx )
      I_Contact( #EstadoVI.Error_Mx )
      I_Contact( #Error_Tx )
      I_Contact( #Centrador_IN )
      Coil( #MA_Cerrar_Centrado )
   END_RUNG
   RUNG wire#powerrail
      Contact( #Mx_ET61 )
   END_RUNG wire#w1
   RUNG wire#powerrail
      Contact( #Mx_ET62 )
      Contact( "OFF" )
   END_RUNG wire#w1
   RUNG wire#powerrail
      Contact( #SimultaneoPaletizado )
      Contact( "ON" )
   END_RUNG wire#w1
   // the same network as SCL:
   #MA_Cerrar_Centrado := (#Mx_ET60 OR #Mx_ET61 OR (#Mx_ET62 AND "OFF") OR (#SimultaneoPaletizado AND "ON")) AND #Permitir_CerrarCentrado AND #EstadoZona.Marcha_CBx AND NOT #EstadoVI.Error_Mx AND NOT #Error_Tx AND NOT #Centrador_IN;
END_REGION

REGION Network 80: SALIDAS - Abrir Centrador
   RUNG wire#powerrail
      I_Contact( #Mx_ET60 )
      I_Contact( #Mx_ET61 )
      wire#w1
      I_Contact( #SimultaneoPaletizado )
      wire#w2
      I_Contact( #Mx_ET62 )
      wire#w3
      Contact( #Permitir_AbrirCentrado )
      Contact( #EstadoZona.Marcha_CBx )
      I_Contact( #EstadoVI.Error_Mx )
      I_Contact( #Error_Tx )
      I_Contact( #Centrador_OUT )
      Coil( #MA_Abrir_Centrado )
   END_RUNG
   RUNG wire#w1
      Contact( "OFF" )
   END_RUNG wire#w2
   RUNG wire#w2
      Contact( "ON" )
   END_RUNG wire#w3
   // the same network as SCL:
   #MA_Abrir_Centrado := NOT #Mx_ET60 AND NOT #Mx_ET61 AND (NOT #SimultaneoPaletizado OR "OFF") AND (NOT #Mx_ET62 OR "ON") AND #Permitir_AbrirCentrado AND #EstadoZona.Marcha_CBx AND NOT #EstadoVI.Error_Mx AND NOT #Error_Tx AND NOT #Centrador_OUT;
END_REGION

REGION Network 81: SALIDAS - Abrir Pala FIja (Recoger)
   RUNG wire#powerrail
      I_Contact( #Mx_ET60 )
      I_Contact( #Mx_ET61 )
      I_Contact( #Mx_ET62 )
      Contact( #Permitir_AbrirPalas )
      Contact( #EstadoZona.Marcha_CBx )
      I_Contact( #EstadoVI.Error_Mx )
      I_Contact( #Error_Tx )
      Contact( #Centrador_OUT )
      I_Contact( #PalaFija_OUT )
      Coil( #MA_Abrir_PalasFija )
   END_RUNG
   // the same network as SCL:
   #MA_Abrir_PalasFija := NOT #Mx_ET60 AND NOT #Mx_ET61 AND NOT #Mx_ET62 AND #Permitir_AbrirPalas AND #EstadoZona.Marcha_CBx AND NOT #EstadoVI.Error_Mx AND NOT #Error_Tx AND #Centrador_OUT AND NOT #PalaFija_OUT;
END_REGION

REGION Network 82: SALIDAS - Cerrar Pala Fija (Extender)
   RUNG wire#powerrail
      Contact( #Mx_ET61 )
      wire#w1
      Contact( #PermisoCierrePalas )
      Contact( #Permitir_CerrarPalas )
      Contact( #EstadoZona.Marcha_CBx )
      I_Contact( #EstadoVI.Error_Mx )
      I_Contact( #Error_Tx )
      Contact( #Centrador_IN )
      I_Contact( #PalaFija_IN )
      Coil( #MA_Cerrar_PalasFija )
   END_RUNG
   RUNG wire#powerrail
      Contact( #Mx_ET62 )
   END_RUNG wire#w1
   // the same network as SCL:
   #MA_Cerrar_PalasFija := (#Mx_ET61 OR #Mx_ET62) AND #PermisoCierrePalas AND #Permitir_CerrarPalas AND #EstadoZona.Marcha_CBx AND NOT #EstadoVI.Error_Mx AND NOT #Error_Tx AND #Centrador_IN AND NOT #PalaFija_IN;
END_REGION

REGION Network 83: SALIDAS - Abrir Pala Movil (Recoger)
   RUNG wire#powerrail
      I_Contact( #Mx_ET60 )
      I_Contact( #Mx_ET61 )
      I_Contact( #Mx_ET62 )
      Contact( #Permitir_AbrirPalas )
      Contact( #EstadoZona.Marcha_CBx )
      I_Contact( #EstadoVI.Error_Mx )
      I_Contact( #Error_Tx )
      Contact( #Centrador_OUT )
      I_Contact( #PalaMovil_OUT )
      Coil( #MA_Abrir_PalasMovil )
   END_RUNG
   // the same network as SCL:
   #MA_Abrir_PalasMovil := NOT #Mx_ET60 AND NOT #Mx_ET61 AND NOT #Mx_ET62 AND #Permitir_AbrirPalas AND #EstadoZona.Marcha_CBx AND NOT #EstadoVI.Error_Mx AND NOT #Error_Tx AND #Centrador_OUT AND NOT #PalaMovil_OUT;
END_REGION

REGION Network 84: SALIDAS - Cerrar Pala Movil (Extender)
   RUNG wire#powerrail
      Contact( #Mx_ET61 )
      wire#w1
      Contact( #PermisoCierrePalas )
      Contact( #Permitir_CerrarPalas )
      Contact( #EstadoZona.Marcha_CBx )
      I_Contact( #EstadoVI.Error_Mx )
      I_Contact( #Error_Tx )
      Contact( #Centrador_IN )
      Contact( #PalaFija_IN )
      I_Contact( #PalaMovil_IN )
      Coil( #MA_Cerrar_PalasMovil )
   END_RUNG
   RUNG wire#powerrail
      Contact( #Mx_ET62 )
   END_RUNG wire#w1
   // the same network as SCL:
   #MA_Cerrar_PalasMovil := (#Mx_ET61 OR #Mx_ET62) AND #PermisoCierrePalas AND #Permitir_CerrarPalas AND #EstadoZona.Marcha_CBx AND NOT #EstadoVI.Error_Mx AND NOT #Error_Tx AND #Centrador_IN AND #PalaFija_IN AND NOT #PalaMovil_IN;
END_REGION

REGION Network 85: SALIDAS - Bajar Mesa Elevadora
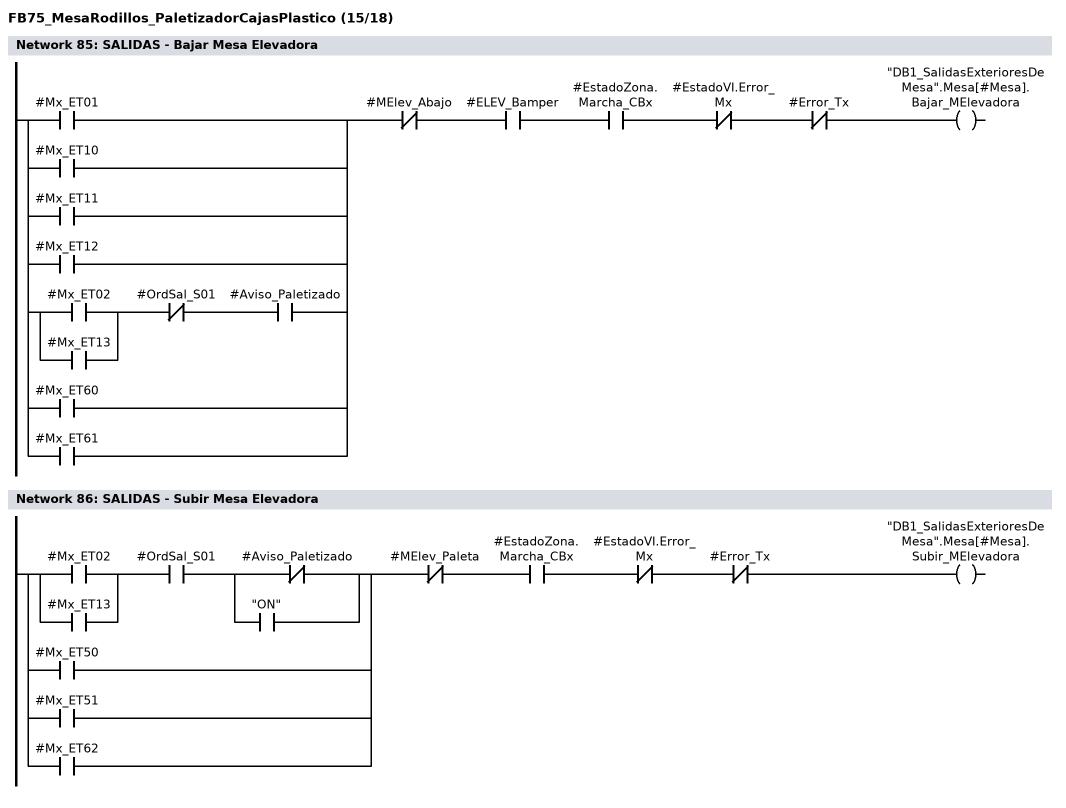
   RUNG wire#powerrail
      Contact( #Mx_ET01 )
      wire#w1
      I_Contact( #MElev_Abajo )
      Contact( #ELEV_Bamper )
      Contact( #EstadoZona.Marcha_CBx )
      I_Contact( #EstadoVI.Error_Mx )
      I_Contact( #Error_Tx )
      Coil( "DB1_SalidasExterioresDeMesa".Mesa[#Mesa].Bajar_MElevadora )
   END_RUNG
   RUNG wire#powerrail
      Contact( #Mx_ET10 )
   END_RUNG wire#w1
   RUNG wire#powerrail
      Contact( #Mx_ET11 )
   END_RUNG wire#w1
   RUNG wire#powerrail
      Contact( #Mx_ET12 )
   END_RUNG wire#w1
   RUNG wire#powerrail
      Contact( #Mx_ET02 )
      wire#w2
      I_Contact( #OrdSal_S01 )
      Contact( #Aviso_Paletizado )
   END_RUNG wire#w1
   RUNG wire#powerrail
      Contact( #Mx_ET13 )
   END_RUNG wire#w2
   RUNG wire#powerrail
      Contact( #Mx_ET60 )
   END_RUNG wire#w1
   RUNG wire#powerrail
      Contact( #Mx_ET61 )
   END_RUNG wire#w1
   // the same network as SCL:
   "DB1_SalidasExterioresDeMesa".Mesa[#Mesa].Bajar_MElevadora := (#Mx_ET01 OR #Mx_ET10 OR #Mx_ET11 OR #Mx_ET12 OR ((#Mx_ET02 OR #Mx_ET13) AND NOT #OrdSal_S01 AND #Aviso_Paletizado) OR #Mx_ET60 OR #Mx_ET61) AND NOT #MElev_Abajo AND #ELEV_Bamper AND #EstadoZona.Marcha_CBx AND NOT #EstadoVI.Error_Mx AND NOT #Error_Tx;
END_REGION

REGION Network 86: SALIDAS - Subir Mesa Elevadora
   RUNG wire#powerrail
      Contact( #Mx_ET02 )
      wire#w1
      Contact( #OrdSal_S01 )
      wire#w2
      I_Contact( #Aviso_Paletizado )
      wire#w3
      I_Contact( #MElev_Paleta )
      Contact( #EstadoZona.Marcha_CBx )
      I_Contact( #EstadoVI.Error_Mx )
      I_Contact( #Error_Tx )
      Coil( "DB1_SalidasExterioresDeMesa".Mesa[#Mesa].Subir_MElevadora )
   END_RUNG
   RUNG wire#powerrail
      Contact( #Mx_ET13 )
   END_RUNG wire#w1
   RUNG wire#w2
      Contact( "ON" )
   END_RUNG wire#w3
   RUNG wire#powerrail
      Contact( #Mx_ET50 )
   END_RUNG wire#w3
   RUNG wire#powerrail
      Contact( #Mx_ET51 )
   END_RUNG wire#w3
   RUNG wire#powerrail
      Contact( #Mx_ET62 )
   END_RUNG wire#w3
   // the same network as SCL:
   "DB1_SalidasExterioresDeMesa".Mesa[#Mesa].Subir_MElevadora := (((#Mx_ET02 OR #Mx_ET13) AND #OrdSal_S01 AND (NOT #Aviso_Paletizado OR "ON")) OR #Mx_ET50 OR #Mx_ET51 OR #Mx_ET62) AND NOT #MElev_Paleta AND #EstadoZona.Marcha_CBx AND NOT #EstadoVI.Error_Mx AND NOT #Error_Tx;
END_REGION

REGION Network 87: ESTADOS DE LA MESA
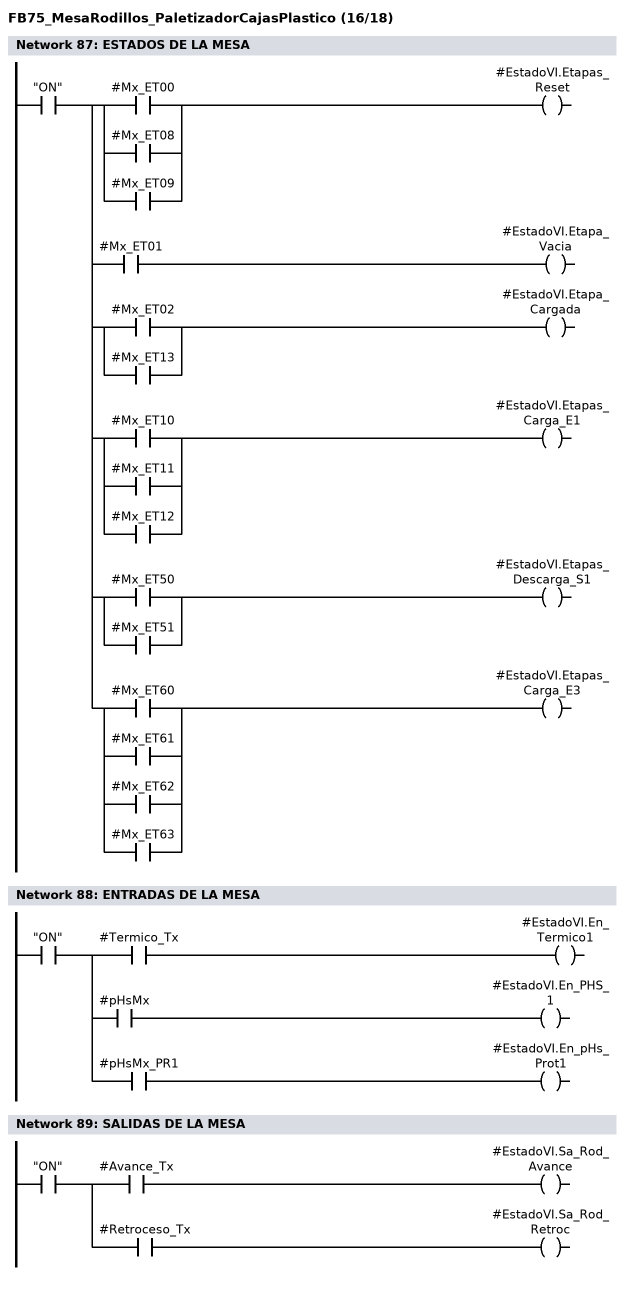
   RUNG wire#powerrail
      Contact( "ON" )
      wire#w1
      Contact( #Mx_ET00 )
      wire#w2
      Coil( #EstadoVI.Etapas_Reset )
   END_RUNG
   RUNG wire#w1
      Contact( #Mx_ET08 )
   END_RUNG wire#w2
   RUNG wire#w1
      Contact( #Mx_ET09 )
   END_RUNG wire#w2
   RUNG wire#w1
      Contact( #Mx_ET01 )
      Coil( #EstadoVI.Etapa_Vacia )
   END_RUNG
   RUNG wire#w1
      Contact( #Mx_ET02 )
      wire#w3
      Coil( #EstadoVI.Etapa_Cargada )
   END_RUNG
   RUNG wire#w1
      Contact( #Mx_ET13 )
   END_RUNG wire#w3
   RUNG wire#w1
      Contact( #Mx_ET10 )
      wire#w4
      Coil( #EstadoVI.Etapas_Carga_E1 )
   END_RUNG
   RUNG wire#w1
      Contact( #Mx_ET11 )
   END_RUNG wire#w4
   RUNG wire#w1
      Contact( #Mx_ET12 )
   END_RUNG wire#w4
   RUNG wire#w1
      Contact( #Mx_ET50 )
      wire#w5
      Coil( #EstadoVI.Etapas_Descarga_S1 )
   END_RUNG
   RUNG wire#w1
      Contact( #Mx_ET51 )
   END_RUNG wire#w5
   RUNG wire#w1
      Contact( #Mx_ET60 )
      wire#w6
      Coil( #EstadoVI.Etapas_Carga_E3 )
   END_RUNG
   RUNG wire#w1
      Contact( #Mx_ET61 )
   END_RUNG wire#w6
   RUNG wire#w1
      Contact( #Mx_ET62 )
   END_RUNG wire#w6
   RUNG wire#w1
      Contact( #Mx_ET63 )
   END_RUNG wire#w6
   // the same network as SCL:
   #EstadoVI.Etapas_Reset := "ON" AND (#Mx_ET00 OR #Mx_ET08 OR #Mx_ET09);
   #EstadoVI.Etapa_Vacia := "ON" AND #Mx_ET01;
   #EstadoVI.Etapa_Cargada := "ON" AND (#Mx_ET02 OR #Mx_ET13);
   #EstadoVI.Etapas_Carga_E1 := "ON" AND (#Mx_ET10 OR #Mx_ET11 OR #Mx_ET12);
   #EstadoVI.Etapas_Descarga_S1 := "ON" AND (#Mx_ET50 OR #Mx_ET51);
   #EstadoVI.Etapas_Carga_E3 := "ON" AND (#Mx_ET60 OR #Mx_ET61 OR #Mx_ET62 OR #Mx_ET63);
END_REGION

REGION Network 88: ENTRADAS DE LA MESA
   RUNG wire#powerrail
      Contact( "ON" )
      wire#w1
      Contact( #Termico_Tx )
      Coil( #EstadoVI.En_Termico1 )
   END_RUNG
   RUNG wire#w1
      Contact( #pHsMx )
      Coil( #EstadoVI.En_PHS_1 )
   END_RUNG
   RUNG wire#w1
      Contact( #pHsMx_PR1 )
      Coil( #EstadoVI.En_pHs_Prot1 )
   END_RUNG
   // the same network as SCL:
   #EstadoVI.En_Termico1 := "ON" AND #Termico_Tx;
   #EstadoVI.En_PHS_1 := "ON" AND #pHsMx;
   #EstadoVI.En_pHs_Prot1 := "ON" AND #pHsMx_PR1;
END_REGION

REGION Network 89: SALIDAS DE LA MESA
   RUNG wire#powerrail
      Contact( "ON" )
      wire#w1
      Contact( #Avance_Tx )
      Coil( #EstadoVI.Sa_Rod_Avance )
   END_RUNG
   RUNG wire#w1
      Contact( #Retroceso_Tx )
      Coil( #EstadoVI.Sa_Rod_Retroc )
   END_RUNG
   // the same network as SCL:
   #EstadoVI.Sa_Rod_Avance := "ON" AND #Avance_Tx;
   #EstadoVI.Sa_Rod_Retroc := "ON" AND #Retroceso_Tx;
END_REGION

REGION Network 90: ESTADOS DE LA MAQUINA (HMI)
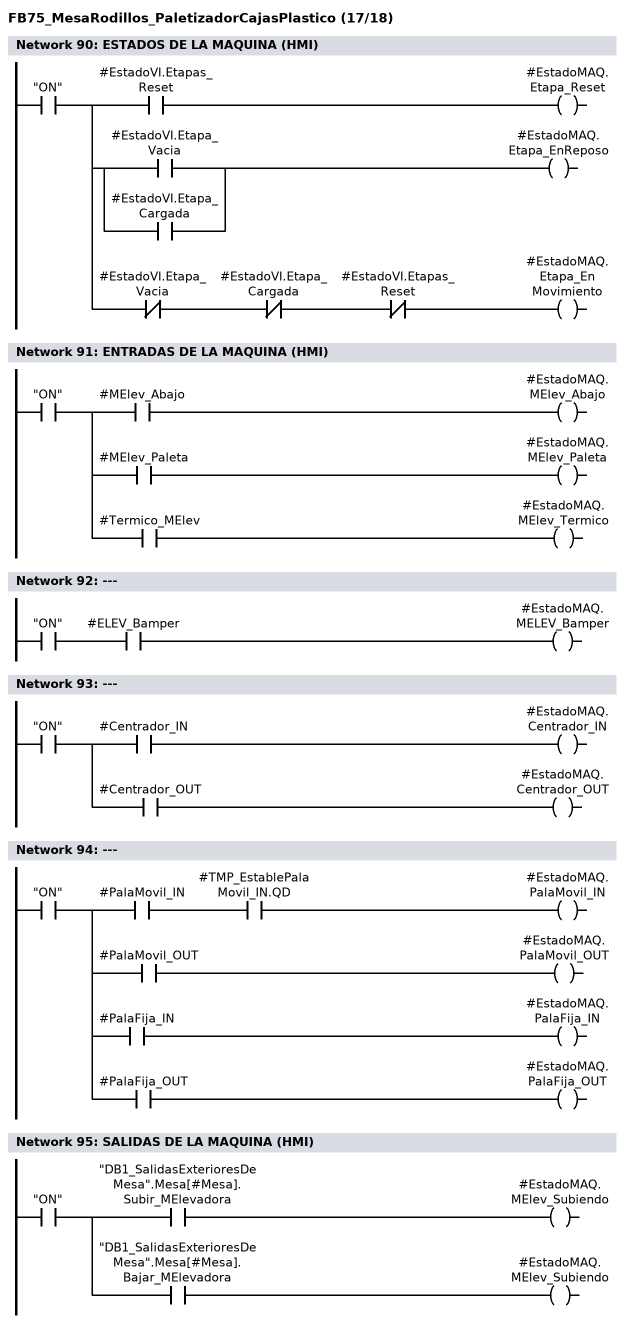
   RUNG wire#powerrail
      Contact( "ON" )
      wire#w1
      Contact( #EstadoVI.Etapas_Reset )
      Coil( #EstadoMAQ.Etapa_Reset )
   END_RUNG
   RUNG wire#w1
      Contact( #EstadoVI.Etapa_Vacia )
      wire#w2
      Coil( #EstadoMAQ.Etapa_EnReposo )
   END_RUNG
   RUNG wire#w1
      Contact( #EstadoVI.Etapa_Cargada )
   END_RUNG wire#w2
   RUNG wire#w1
      I_Contact( #EstadoVI.Etapa_Vacia )
      I_Contact( #EstadoVI.Etapa_Cargada )
      I_Contact( #EstadoVI.Etapas_Reset )
      Coil( #EstadoMAQ.Etapa_EnMovimiento )
   END_RUNG
   // the same network as SCL:
   #EstadoMAQ.Etapa_Reset := "ON" AND #EstadoVI.Etapas_Reset;
   #EstadoMAQ.Etapa_EnReposo := "ON" AND (#EstadoVI.Etapa_Vacia OR #EstadoVI.Etapa_Cargada);
   #EstadoMAQ.Etapa_EnMovimiento := "ON" AND NOT #EstadoVI.Etapa_Vacia AND NOT #EstadoVI.Etapa_Cargada AND NOT #EstadoVI.Etapas_Reset;
END_REGION

REGION Network 91: ENTRADAS DE LA MAQUINA (HMI)
   RUNG wire#powerrail
      Contact( "ON" )
      wire#w1
      Contact( #MElev_Abajo )
      Coil( #EstadoMAQ.MElev_Abajo )
   END_RUNG
   RUNG wire#w1
      Contact( #MElev_Paleta )
      Coil( #EstadoMAQ.MElev_Paleta )
   END_RUNG
   RUNG wire#w1
      Contact( #Termico_MElev )
      Coil( #EstadoMAQ.MElev_Termico )
   END_RUNG
   // the same network as SCL:
   #EstadoMAQ.MElev_Abajo := "ON" AND #MElev_Abajo;
   #EstadoMAQ.MElev_Paleta := "ON" AND #MElev_Paleta;
   #EstadoMAQ.MElev_Termico := "ON" AND #Termico_MElev;
END_REGION

REGION Network 92: ---
   RUNG wire#powerrail
      Contact( "ON" )
      Contact( #ELEV_Bamper )
      Coil( #EstadoMAQ.MELEV_Bamper )
   END_RUNG
   // the same network as SCL:
   #EstadoMAQ.MELEV_Bamper := "ON" AND #ELEV_Bamper;
END_REGION

REGION Network 93: ---
   RUNG wire#powerrail
      Contact( "ON" )
      wire#w1
      Contact( #Centrador_IN )
      Coil( #EstadoMAQ.Centrador_IN )
   END_RUNG
   RUNG wire#w1
      Contact( #Centrador_OUT )
      Coil( #EstadoMAQ.Centrador_OUT )
   END_RUNG
   // the same network as SCL:
   #EstadoMAQ.Centrador_IN := "ON" AND #Centrador_IN;
   #EstadoMAQ.Centrador_OUT := "ON" AND #Centrador_OUT;
END_REGION

REGION Network 94: ---
   RUNG wire#powerrail
      Contact( "ON" )
      wire#w1
      Contact( #PalaMovil_IN )
      Contact( #TMP_EstablePalaMovil_IN.QD )
      Coil( #EstadoMAQ.PalaMovil_IN )
   END_RUNG
   RUNG wire#w1
      Contact( #PalaMovil_OUT )
      Coil( #EstadoMAQ.PalaMovil_OUT )
   END_RUNG
   RUNG wire#w1
      Contact( #PalaFija_IN )
      Coil( #EstadoMAQ.PalaFija_IN )
   END_RUNG
   RUNG wire#w1
      Contact( #PalaFija_OUT )
      Coil( #EstadoMAQ.PalaFija_OUT )
   END_RUNG
   // the same network as SCL:
   #EstadoMAQ.PalaMovil_IN := "ON" AND #PalaMovil_IN AND #TMP_EstablePalaMovil_IN.QD;
   #EstadoMAQ.PalaMovil_OUT := "ON" AND #PalaMovil_OUT;
   #EstadoMAQ.PalaFija_IN := "ON" AND #PalaFija_IN;
   #EstadoMAQ.PalaFija_OUT := "ON" AND #PalaFija_OUT;
END_REGION

REGION Network 95: SALIDAS DE LA MAQUINA (HMI)
   RUNG wire#powerrail
      Contact( "ON" )
      wire#w1
      Contact( "DB1_SalidasExterioresDeMesa".Mesa[#Mesa].Subir_MElevadora )
      Coil( #EstadoMAQ.MElev_Subiendo )
   END_RUNG
   RUNG wire#w1
      Contact( "DB1_SalidasExterioresDeMesa".Mesa[#Mesa].Bajar_MElevadora )
      Coil( #EstadoMAQ.MElev_Subiendo )
   END_RUNG
   // the same network as SCL:
   #EstadoMAQ.MElev_Subiendo := "ON" AND "DB1_SalidasExterioresDeMesa".Mesa[#Mesa].Subir_MElevadora;
   #EstadoMAQ.MElev_Subiendo := "ON" AND "DB1_SalidasExterioresDeMesa".Mesa[#Mesa].Bajar_MElevadora;
END_REGION

REGION Network 96: ---
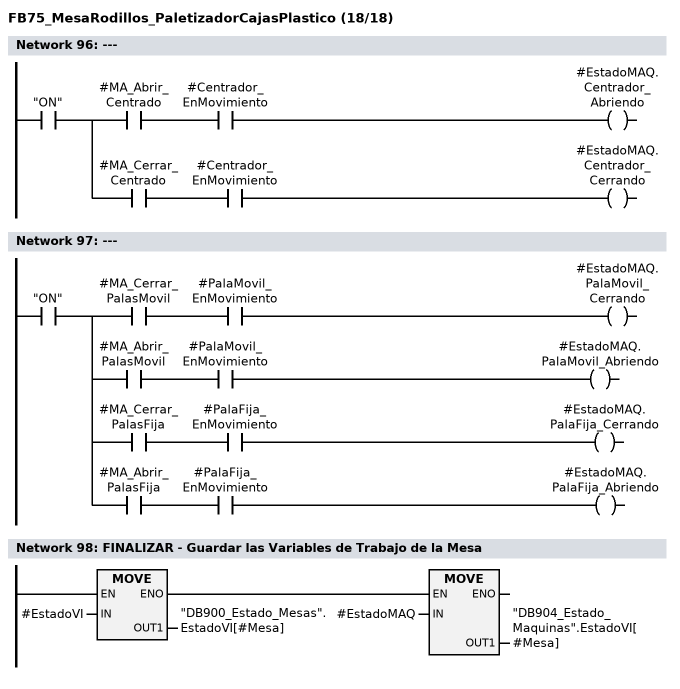
   RUNG wire#powerrail
      Contact( "ON" )
      wire#w1
      Contact( #MA_Abrir_Centrado )
      Contact( #Centrador_EnMovimiento )
      Coil( #EstadoMAQ.Centrador_Abriendo )
   END_RUNG
   RUNG wire#w1
      Contact( #MA_Cerrar_Centrado )
      Contact( #Centrador_EnMovimiento )
      Coil( #EstadoMAQ.Centrador_Cerrando )
   END_RUNG
   // the same network as SCL:
   #EstadoMAQ.Centrador_Abriendo := "ON" AND #MA_Abrir_Centrado AND #Centrador_EnMovimiento;
   #EstadoMAQ.Centrador_Cerrando := "ON" AND #MA_Cerrar_Centrado AND #Centrador_EnMovimiento;
END_REGION

REGION Network 97: ---
   RUNG wire#powerrail
      Contact( "ON" )
      wire#w1
      Contact( #MA_Cerrar_PalasMovil )
      Contact( #PalaMovil_EnMovimiento )
      Coil( #EstadoMAQ.PalaMovil_Cerrando )
   END_RUNG
   RUNG wire#w1
      Contact( #MA_Abrir_PalasMovil )
      Contact( #PalaMovil_EnMovimiento )
      Coil( #EstadoMAQ.PalaMovil_Abriendo )
   END_RUNG
   RUNG wire#w1
      Contact( #MA_Cerrar_PalasFija )
      Contact( #PalaFija_EnMovimiento )
      Coil( #EstadoMAQ.PalaFija_Cerrando )
   END_RUNG
   RUNG wire#w1
      Contact( #MA_Abrir_PalasFija )
      Contact( #PalaFija_EnMovimiento )
      Coil( #EstadoMAQ.PalaFija_Abriendo )
   END_RUNG
   // the same network as SCL:
   #EstadoMAQ.PalaMovil_Cerrando := "ON" AND #MA_Cerrar_PalasMovil AND #PalaMovil_EnMovimiento;
   #EstadoMAQ.PalaMovil_Abriendo := "ON" AND #MA_Abrir_PalasMovil AND #PalaMovil_EnMovimiento;
   #EstadoMAQ.PalaFija_Cerrando := "ON" AND #MA_Cerrar_PalasFija AND #PalaFija_EnMovimiento;
   #EstadoMAQ.PalaFija_Abriendo := "ON" AND #MA_Abrir_PalasFija AND #PalaFija_EnMovimiento;
END_REGION

REGION Network 98: FINALIZAR - Guardar las Variables de Trabajo de la Mesa
   RUNG wire#powerrail
      Move(in := #EstadoVI, out1 => "DB900_Estado_Mesas".EstadoVI[#Mesa])
      Move(in := #EstadoMAQ, out1 => "DB904_Estado_Maquinas".EstadoVI[#Mesa])
   END_RUNG
   // the same network as SCL:
   "DB900_Estado_Mesas".EstadoVI[#Mesa] := #EstadoVI;
   "DB904_Estado_Maquinas".EstadoVI[#Mesa] := #EstadoMAQ;
END_REGION
END_FUNCTION_BLOCK
